Yaskawa INFORM job: CONTOUR.JBI

/JOB
//NAME CONTOUR
//POS
///NPOS 1076,0,0,0,0,0
///TOOL 0
///POSTYPE PULSE
///PULSE
C00000=-2822,58859,-1118,-1041,-34109,-89
C00001=-2184,59252,651,-1119,-34320,-350
C00002=-2184,59252,-549,-1119,-34320,-350
C00003=-2209,59236,-572,-1116,-34311,-340
C00004=-2228,59203,-624,-1114,-34290,-332
C00005=-2241,59164,-682,-1113,-34266,-326
C00006=-2250,59123,-744,-1112,-34241,-322
C00007=-2256,59080,-810,-1112,-34215,-319
C00008=-2257,59034,-879,-1113,-34187,-318
C00009=-2256,58989,-948,-1113,-34159,-318
C00010=-2251,58945,-1015,-1115,-34132,-319
C00011=-2245,58902,-1080,-1116,-34106,-321
C00012=-2233,58862,-1139,-1118,-34082,-326
C00013=-2213,58831,-1186,-1122,-34063,-333
C00014=-2187,58817,-1207,-1125,-34055,-343
C00015=-2161,58829,-1188,-1128,-34062,-354
C00016=-2142,58860,-1141,-1130,-34081,-362
C00017=-2133,58899,-1082,-1131,-34105,-367
C00018=-2146,58931,-1034,-1129,-34125,-362
C00019=-2150,58886,-1101,-1129,-34097,-359
C00020=-2165,58851,-1155,-1127,-34076,-353
C00021=-2191,58837,-1177,-1124,-34067,-342
C00022=-2215,58858,-1145,-1121,-34080,-333
C00023=-2231,58895,-1089,-1118,-34102,-327
C00024=-2239,58937,-1026,-1116,-34128,-324
C00025=-2243,58981,-959,-1115,-34155,-323
C00026=-2246,59026,-891,-1114,-34182,-322
C00027=-2245,59072,-822,-1113,-34210,-323
C00028=-2239,59115,-756,-1114,-34237,-326
C00029=-2230,59156,-694,-1114,-34261,-331
C00030=-2215,59193,-638,-1115,-34284,-337
C00031=-2195,59225,-590,-1118,-34304,-346
C00032=-2168,59227,-586,-1121,-34305,-357
C00033=-2143,59211,-610,-1125,-34296,-367
C00034=-2134,59169,-673,-1126,-34270,-369
C00035=-2128,59126,-737,-1128,-34244,-371
C00036=-2125,59081,-805,-1129,-34217,-372
C00037=-2109,59103,-772,-1131,-34230,-379
C00038=-2115,59146,-707,-1129,-34256,-377
C00039=-2123,59188,-644,-1128,-34282,-374
C00040=-2131,59230,-580,-1126,-34307,-372
C00041=-2155,59248,-554,-1122,-34318,-362
C00042=-2184,59252,-549,-1119,-34320,-350
C00043=-2184,59252,651,-1119,-34320,-350
C00044=-1874,59033,327,-1163,-34189,-472
C00045=-1874,59033,-873,-1163,-34189,-472
C00046=-1891,59025,-886,-1161,-34184,-465
C00047=-1906,59007,-912,-1159,-34173,-459
C00048=-1916,58983,-950,-1158,-34158,-455
C00049=-1926,58964,-979,-1157,-34146,-450
C00050=-1930,58992,-936,-1156,-34164,-449
C00051=-1936,59020,-895,-1155,-34180,-447
C00052=-1949,59030,-879,-1153,-34186,-442
C00053=-1949,59002,-922,-1153,-34169,-442
C00054=-1942,58975,-962,-1155,-34153,-444
C00055=-1936,58948,-1003,-1156,-34136,-446
C00056=-1933,58919,-1047,-1157,-34119,-447
C00057=-1930,58890,-1091,-1158,-34101,-448
C00058=-1928,58860,-1136,-1158,-34083,-448
C00059=-1925,58831,-1180,-1159,-34065,-449
C00060=-1914,58811,-1211,-1161,-34052,-453
C00061=-1907,58835,-1174,-1162,-34067,-456
C00062=-1911,58864,-1130,-1161,-34085,-455
C00063=-1912,58893,-1086,-1160,-34103,-455
C00064=-1913,58924,-1039,-1159,-34122,-455
C00065=-1911,58952,-997,-1159,-34139,-457
C00066=-1904,58978,-957,-1160,-34155,-460
C00067=-1892,59001,-922,-1161,-34169,-465
C00068=-1875,59009,-909,-1163,-34175,-472
C00069=-1858,59003,-918,-1165,-34171,-479
C00070=-1844,58981,-950,-1167,-34158,-484
C00071=-1834,58957,-988,-1169,-34142,-487
C00072=-1828,58930,-1029,-1170,-34126,-490
C00073=-1822,58902,-1070,-1172,-34109,-492
C00074=-1819,58873,-1114,-1173,-34092,-493
C00075=-1818,58843,-1160,-1173,-34073,-493
C00076=-1806,58826,-1186,-1175,-34063,-497
C00077=-1798,58850,-1149,-1176,-34078,-500
C00078=-1803,58878,-1107,-1175,-34095,-499
C00079=-1810,58905,-1066,-1173,-34111,-497
C00080=-1814,58933,-1023,-1172,-34128,-495
C00081=-1821,58960,-983,-1171,-34145,-493
C00082=-1830,58986,-944,-1169,-34160,-490
C00083=-1841,59009,-908,-1167,-34175,-485
C00084=-1856,59028,-880,-1165,-34186,-480
C00085=-1874,59033,-873,-1163,-34189,-472
C00086=-1874,59033,327,-1163,-34189,-472
C00087=-1240,59056,376,-1245,-34208,-728
C00088=-1240,59056,-824,-1245,-34208,-728
C00089=-1239,59026,-870,-1246,-34189,-728
C00090=-1230,58999,-911,-1247,-34173,-731
C00091=-1224,58970,-954,-1249,-34155,-733
C00092=-1220,58941,-999,-1250,-34137,-734
C00093=-1215,58911,-1044,-1251,-34119,-736
C00094=-1214,58881,-1090,-1252,-34100,-736
C00095=-1216,58849,-1139,-1252,-34081,-735
C00096=-1220,58819,-1183,-1252,-34062,-733
C00097=-1232,58796,-1220,-1251,-34048,-728
C00098=-1251,58791,-1227,-1248,-34045,-720
C00099=-1268,58804,-1208,-1246,-34053,-713
C00100=-1284,58821,-1182,-1244,-34063,-707
C00101=-1298,58844,-1148,-1241,-34077,-702
C00102=-1307,58870,-1108,-1240,-34093,-698
C00103=-1313,58899,-1064,-1238,-34111,-696
C00104=-1318,58929,-1019,-1237,-34129,-695
C00105=-1321,58959,-973,-1236,-34148,-694
C00106=-1321,58991,-925,-1236,-34167,-694
C00107=-1335,59000,-910,-1234,-34173,-689
C00108=-1336,58972,-953,-1234,-34156,-688
C00109=-1333,58942,-999,-1235,-34137,-689
C00110=-1329,58912,-1045,-1236,-34119,-690
C00111=-1325,58882,-1090,-1237,-34101,-691
C00112=-1319,58854,-1133,-1238,-34083,-693
C00113=-1307,58828,-1172,-1240,-34067,-698
C00114=-1294,58805,-1207,-1242,-34053,-703
C00115=-1278,58788,-1233,-1245,-34043,-709
C00116=-1261,58774,-1254,-1247,-34034,-715
C00117=-1243,58771,-1258,-1250,-34032,-723
C00118=-1224,58777,-1248,-1252,-34036,-730
C00119=-1211,58799,-1214,-1253,-34050,-736
C00120=-1204,58827,-1171,-1254,-34067,-739
C00121=-1202,58859,-1123,-1254,-34087,-740
C00122=-1201,58890,-1075,-1253,-34106,-741
C00123=-1204,58920,-1029,-1252,-34125,-740
C00124=-1208,58951,-983,-1251,-34143,-739
C00125=-1213,58980,-939,-1250,-34161,-738
C00126=-1219,59008,-896,-1249,-34179,-736
C00127=-1227,59036,-854,-1247,-34196,-733
C00128=-1240,59056,-824,-1245,-34208,-728
C00129=-1240,59056,376,-1245,-34208,-728
C00130=-2046,59034,324,-1140,-34188,-403
C00131=-2046,59034,-876,-1140,-34188,-403
C00132=-2039,59033,-876,-1141,-34188,-406
C00133=-2033,59026,-888,-1142,-34183,-408
C00134=-2027,59017,-900,-1143,-34178,-411
C00135=-2021,59011,-910,-1144,-34174,-413
C00136=-2016,59002,-923,-1145,-34169,-415
C00137=-2013,58991,-940,-1145,-34162,-416
C00138=-2012,58979,-958,-1145,-34155,-416
C00139=-2012,58967,-976,-1146,-34148,-416
C00140=-2014,58955,-994,-1146,-34141,-415
C00141=-2013,58943,-1012,-1146,-34133,-415
C00142=-2014,58931,-1030,-1146,-34126,-415
C00143=-2015,58918,-1050,-1146,-34118,-414
C00144=-2016,58906,-1068,-1146,-34110,-414
C00145=-2017,58894,-1086,-1146,-34103,-413
C00146=-2020,58883,-1104,-1146,-34096,-412
C00147=-2024,58873,-1119,-1146,-34090,-410
C00148=-2029,58864,-1133,-1145,-34084,-408
C00149=-2035,58856,-1144,-1145,-34080,-405
C00150=-2042,58853,-1149,-1144,-34078,-402
C00151=-2050,58852,-1151,-1143,-34077,-399
C00152=-2057,58856,-1144,-1142,-34080,-396
C00153=-2064,58859,-1140,-1141,-34081,-394
C00154=-2070,58867,-1128,-1140,-34086,-391
C00155=-2076,58874,-1118,-1139,-34090,-389
C00156=-2081,58884,-1103,-1138,-34097,-387
C00157=-2084,58895,-1086,-1137,-34103,-386
C00158=-2087,58906,-1069,-1137,-34110,-385
C00159=-2087,58919,-1051,-1137,-34118,-385
C00160=-2088,58931,-1032,-1136,-34125,-385
C00161=-2087,58943,-1014,-1136,-34132,-385
C00162=-2086,58955,-996,-1136,-34140,-386
C00163=-2083,58966,-979,-1136,-34146,-387
C00164=-2080,58977,-963,-1137,-34153,-389
C00165=-2078,58988,-946,-1137,-34160,-390
C00166=-2074,58998,-930,-1137,-34166,-392
C00167=-2070,59007,-916,-1137,-34172,-393
C00168=-2066,59017,-901,-1138,-34178,-395
C00169=-2060,59025,-890,-1139,-34183,-398
C00170=-2053,59029,-883,-1139,-34185,-400
C00171=-2046,59034,-876,-1140,-34188,-403
C00172=-2046,59034,324,-1140,-34188,-403
C00173=-1405,59028,330,-1224,-34190,-661
C00174=-1405,59028,-870,-1224,-34190,-661
C00175=-1398,59001,-912,-1226,-34173,-664
C00176=-1386,58977,-947,-1228,-34159,-668
C00177=-1375,58952,-985,-1229,-34143,-672
C00178=-1368,58924,-1027,-1231,-34126,-674
C00179=-1363,58896,-1070,-1232,-34109,-676
C00180=-1359,58866,-1115,-1233,-34090,-677
C00181=-1361,58835,-1163,-1233,-34071,-676
C00182=-1371,58810,-1201,-1232,-34056,-672
C00183=-1389,58802,-1213,-1230,-34051,-664
C00184=-1407,58808,-1204,-1228,-34054,-657
C00185=-1423,58827,-1176,-1225,-34066,-651
C00186=-1433,58852,-1138,-1223,-34081,-647
C00187=-1442,58879,-1098,-1222,-34098,-644
C00188=-1445,58909,-1052,-1221,-34116,-643
C00189=-1443,58939,-1006,-1221,-34135,-645
C00190=-1434,58965,-966,-1221,-34151,-649
C00191=-1419,58984,-938,-1223,-34162,-655
C00192=-1405,58980,-943,-1225,-34160,-661
C00193=-1415,59003,-908,-1223,-34174,-657
C00194=-1433,58997,-917,-1221,-34170,-649
C00195=-1448,58976,-949,-1219,-34158,-643
C00196=-1456,58950,-990,-1219,-34141,-640
C00197=-1460,58920,-1035,-1219,-34123,-638
C00198=-1459,58889,-1082,-1220,-34104,-638
C00199=-1453,58861,-1125,-1221,-34086,-640
C00200=-1442,58835,-1164,-1223,-34071,-643
C00201=-1432,58810,-1203,-1224,-34055,-647
C00202=-1417,58791,-1231,-1227,-34044,-653
C00203=-1399,58782,-1244,-1229,-34038,-660
C00204=-1380,58781,-1245,-1232,-34038,-668
C00205=-1362,58792,-1229,-1234,-34044,-675
C00206=-1352,58816,-1192,-1235,-34059,-680
C00207=-1347,58845,-1147,-1235,-34077,-682
C00208=-1348,58876,-1100,-1234,-34097,-682
C00209=-1352,58906,-1055,-1233,-34115,-681
C00210=-1358,58934,-1013,-1232,-34132,-679
C00211=-1365,58961,-971,-1230,-34149,-676
C00212=-1376,58986,-933,-1229,-34164,-672
C00213=-1389,59010,-897,-1226,-34179,-667
C00214=-1405,59028,-870,-1224,-34190,-661
C00215=-1405,59028,330,-1224,-34190,-661
C00216=-2050,59056,358,-1139,-34202,-402
C00217=-2050,59056,-842,-1139,-34202,-402
C00218=-2062,59047,-855,-1138,-34196,-397
C00219=-2072,59034,-875,-1137,-34188,-393
C00220=-2082,59018,-900,-1136,-34179,-389
C00221=-2088,59000,-927,-1135,-34168,-386
C00222=-2094,58982,-956,-1135,-34156,-383
C00223=-2098,58962,-986,-1135,-34144,-381
C00224=-2101,58941,-1017,-1135,-34131,-380
C00225=-2100,58919,-1050,-1135,-34118,-380
C00226=-2097,58899,-1081,-1136,-34105,-381
C00227=-2093,58879,-1111,-1137,-34093,-382
C00228=-2086,58861,-1139,-1138,-34082,-385
C00229=-2075,58850,-1155,-1139,-34075,-389
C00230=-2064,58840,-1170,-1141,-34070,-394
C00231=-2051,58834,-1178,-1143,-34066,-399
C00232=-2037,58836,-1176,-1145,-34067,-404
C00233=-2025,58842,-1165,-1146,-34071,-409
C00234=-2014,58856,-1144,-1147,-34080,-414
C00235=-2008,58874,-1116,-1148,-34091,-416
C00236=-2004,58894,-1086,-1148,-34103,-418
C00237=-2002,58916,-1053,-1148,-34116,-419
C00238=-1995,58905,-1069,-1149,-34110,-422
C00239=-1990,58886,-1098,-1150,-34098,-424
C00240=-1986,58866,-1128,-1151,-34086,-425
C00241=-1983,58846,-1159,-1152,-34074,-426
C00242=-1976,58829,-1185,-1153,-34063,-429
C00243=-1963,58829,-1185,-1154,-34063,-434
C00244=-1965,58848,-1156,-1154,-34075,-433
C00245=-1972,58866,-1128,-1153,-34086,-431
C00246=-1976,58886,-1098,-1152,-34098,-430
C00247=-1980,58906,-1068,-1151,-34110,-428
C00248=-1984,58926,-1038,-1150,-34123,-427
C00249=-1989,58945,-1009,-1149,-34134,-425
C00250=-1992,58966,-978,-1148,-34147,-424
C00251=-1995,58986,-947,-1148,-34159,-423
C00252=-1999,59006,-917,-1147,-34171,-422
C00253=-2004,59025,-888,-1146,-34183,-420
C00254=-2016,59026,-887,-1144,-34184,-415
C00255=-2026,59042,-863,-1143,-34193,-411
C00256=-2036,59055,-843,-1141,-34201,-407
C00257=-2050,59056,-842,-1139,-34202,-402
C00258=-2050,59056,358,-1139,-34202,-402
C00259=-1609,59068,387,-1197,-34213,-579
C00260=-1609,59068,-813,-1197,-34213,-579
C00261=-1614,59016,-893,-1197,-34180,-577
C00262=-1610,58960,-979,-1199,-34146,-578
C00263=-1598,58908,-1057,-1201,-34114,-582
C00264=-1580,58861,-1128,-1204,-34086,-588
C00265=-1547,58852,-1140,-1209,-34080,-602
C00266=-1529,58898,-1070,-1210,-34109,-609
C00267=-1527,58953,-987,-1209,-34143,-611
C00268=-1514,58951,-990,-1211,-34141,-616
C00269=-1493,58905,-1060,-1215,-34113,-624
C00270=-1475,58856,-1132,-1218,-34084,-631
C00271=-1464,58804,-1212,-1220,-34051,-634
C00272=-1466,58747,-1298,-1221,-34016,-633
C00273=-1481,58698,-1373,-1220,-33986,-626
C00274=-1503,58656,-1438,-1218,-33960,-617
C00275=-1534,58636,-1468,-1214,-33948,-604
C00276=-1565,58661,-1431,-1210,-33963,-592
C00277=-1589,58705,-1365,-1206,-33990,-582
C00278=-1608,58752,-1293,-1202,-34019,-576
C00279=-1616,58761,-1281,-1201,-34024,-573
C00280=-1600,58711,-1356,-1204,-33993,-578
C00281=-1579,58665,-1425,-1208,-33965,-586
C00282=-1553,58628,-1481,-1212,-33943,-596
C00283=-1518,58620,-1493,-1216,-33938,-610
C00284=-1488,58646,-1453,-1220,-33954,-623
C00285=-1467,58690,-1385,-1222,-33981,-632
C00286=-1453,58740,-1309,-1223,-34012,-638
C00287=-1451,58795,-1225,-1222,-34046,-640
C00288=-1458,58849,-1143,-1220,-34079,-637
C00289=-1474,58899,-1068,-1217,-34109,-632
C00290=-1493,58945,-998,-1214,-34138,-625
C00291=-1515,58990,-930,-1210,-34166,-616
C00292=-1534,59037,-860,-1207,-34194,-610
C00293=-1544,59007,-905,-1206,-34176,-605
C00294=-1538,58952,-989,-1208,-34142,-606
C00295=-1540,58896,-1073,-1209,-34108,-605
C00296=-1564,58871,-1113,-1206,-34092,-595
C00297=-1585,58912,-1050,-1203,-34117,-587
C00298=-1595,58965,-970,-1200,-34150,-584
C00299=-1599,59022,-884,-1199,-34184,-583
C00300=-1609,59068,-813,-1197,-34213,-579
C00301=-1609,59068,387,-1197,-34213,-579
C00302=-3014,58953,182,-1015,-34132,-13
C00303=-3014,58953,-1018,-1015,-34132,-13
C00304=-3024,58937,-1043,-1014,-34122,-9
C00305=-3030,58917,-1073,-1013,-34110,-6
C00306=-3034,58895,-1106,-1013,-34097,-4
C00307=-3037,58873,-1140,-1013,-34083,-3
C00308=-3040,58850,-1174,-1013,-34070,-1
C00309=-3044,58828,-1207,-1013,-34057,1
C00310=-3046,58805,-1242,-1013,-34043,2
C00311=-3047,58782,-1277,-1013,-34028,3
C00312=-3049,58758,-1312,-1013,-34014,4
C00313=-3050,58734,-1349,-1013,-34000,4
C00314=-3050,58712,-1383,-1013,-33986,5
C00315=-3048,58689,-1417,-1014,-33972,4
C00316=-3047,58666,-1452,-1015,-33958,4
C00317=-3043,58644,-1484,-1015,-33945,3
C00318=-3037,58624,-1515,-1016,-33933,1
C00319=-3031,58604,-1545,-1018,-33921,-2
C00320=-3021,58586,-1571,-1019,-33910,-5
C00321=-3009,58576,-1587,-1021,-33904,-10
C00322=-2996,58566,-1601,-1023,-33898,-15
C00323=-2983,58561,-1609,-1025,-33895,-21
C00324=-2970,58570,-1595,-1026,-33901,-26
C00325=-2959,58584,-1573,-1027,-33909,-30
C00326=-2955,58606,-1541,-1028,-33922,-32
C00327=-2952,58628,-1507,-1028,-33936,-34
C00328=-2946,58649,-1475,-1028,-33948,-36
C00329=-2946,58673,-1439,-1028,-33963,-37
C00330=-2948,58696,-1405,-1027,-33977,-36
C00331=-2950,58719,-1370,-1027,-33991,-36
C00332=-2952,58740,-1339,-1026,-34003,-35
C00333=-2953,58763,-1303,-1025,-34018,-35
C00334=-2957,58785,-1271,-1025,-34031,-34
C00335=-2961,58806,-1239,-1024,-34044,-32
C00336=-2965,58828,-1206,-1023,-34057,-31
C00337=-2969,58849,-1174,-1022,-34070,-29
C00338=-2972,58871,-1141,-1021,-34083,-28
C00339=-2983,58885,-1120,-1020,-34091,-24
C00340=-2991,58903,-1093,-1018,-34102,-21
C00341=-2996,58924,-1061,-1017,-34115,-20
C00342=-3001,58944,-1032,-1016,-34127,-18
C00343=-3014,58953,-1018,-1015,-34132,-13
C00344=-3014,58953,182,-1015,-34132,-13
C00345=-2663,58940,170,-1061,-34127,-154
C00346=-2663,58940,-1030,-1061,-34127,-154
C00347=-2675,58925,-1053,-1060,-34118,-149
C00348=-2682,58905,-1084,-1059,-34105,-145
C00349=-2691,58886,-1113,-1058,-34094,-142
C00350=-2696,58863,-1147,-1058,-34080,-140
C00351=-2699,58840,-1183,-1058,-34065,-138
C00352=-2702,58816,-1219,-1058,-34051,-137
C00353=-2705,58792,-1254,-1058,-34037,-135
C00354=-2707,58769,-1290,-1058,-34022,-134
C00355=-2709,58744,-1327,-1058,-34007,-133
C00356=-2710,58719,-1365,-1058,-33992,-132
C00357=-2710,58693,-1404,-1058,-33977,-132
C00358=-2707,58671,-1438,-1059,-33963,-133
C00359=-2700,58649,-1470,-1060,-33950,-135
C00360=-2696,58627,-1504,-1061,-33936,-137
C00361=-2690,58605,-1537,-1062,-33923,-139
C00362=-2684,58584,-1569,-1064,-33910,-141
C00363=-2677,58563,-1601,-1065,-33897,-143
C00364=-2668,58543,-1630,-1066,-33885,-147
C00365=-2658,58524,-1659,-1068,-33874,-150
C00366=-2645,58514,-1674,-1070,-33868,-156
C00367=-2631,58520,-1665,-1072,-33871,-161
C00368=-2623,58540,-1635,-1072,-33883,-165
C00369=-2617,58561,-1603,-1073,-33896,-168
C00370=-2611,58582,-1570,-1073,-33910,-170
C00371=-2608,58606,-1534,-1073,-33924,-172
C00372=-2608,58631,-1496,-1073,-33939,-172
C00373=-2607,58657,-1457,-1073,-33955,-173
C00374=-2608,58681,-1420,-1072,-33970,-173
C00375=-2609,58706,-1383,-1072,-33985,-173
C00376=-2611,58730,-1347,-1071,-33999,-172
C00377=-2614,58753,-1312,-1070,-34013,-171
C00378=-2617,58776,-1277,-1069,-34027,-170
C00379=-2620,58799,-1242,-1069,-34041,-169
C00380=-2625,58822,-1208,-1068,-34055,-168
C00381=-2628,58845,-1174,-1067,-34069,-167
C00382=-2632,58868,-1139,-1066,-34083,-165
C00383=-2638,58889,-1107,-1065,-34096,-163
C00384=-2644,58911,-1075,-1064,-34109,-161
C00385=-2650,58932,-1042,-1063,-34122,-159
C00386=-2663,58940,-1030,-1061,-34127,-154
C00387=-2663,58940,170,-1061,-34127,-154
C00388=-2757,59223,596,-1044,-34298,-119
C00389=-2757,59223,-604,-1044,-34298,-119
C00390=-2693,59208,-626,-1053,-34290,-145
C00391=-2630,59182,-664,-1061,-34274,-170
C00392=-2574,59133,-737,-1069,-34245,-192
C00393=-2526,59062,-843,-1077,-34202,-210
C00394=-2480,58986,-957,-1084,-34156,-228
C00395=-2446,58899,-1088,-1090,-34103,-240
C00396=-2419,58806,-1228,-1095,-34047,-250
C00397=-2407,58704,-1382,-1098,-33985,-254
C00398=-2398,58601,-1538,-1101,-33922,-256
C00399=-2407,58496,-1697,-1101,-33858,-251
C00400=-2428,58399,-1844,-1100,-33799,-241
C00401=-2458,58309,-1981,-1098,-33744,-228
C00402=-2493,58223,-2111,-1094,-33691,-213
C00403=-2541,58152,-2220,-1089,-33648,-193
C00404=-2597,58101,-2298,-1083,-33616,-170
C00405=-2656,58061,-2359,-1075,-33592,-146
C00406=-2720,58047,-2380,-1067,-33584,-120
C00407=-2787,58043,-2387,-1058,-33581,-93
C00408=-2853,58050,-2378,-1049,-33585,-66
C00409=-2917,58074,-2342,-1041,-33600,-41
C00410=-2978,58104,-2299,-1032,-33618,-17
C00411=-3037,58144,-2238,-1024,-33642,6
C00412=-3091,58201,-2154,-1016,-33677,27
C00413=-3135,58277,-2039,-1009,-33723,44
C00414=-3171,58365,-1907,-1003,-33776,57
C00415=-3195,58460,-1765,-998,-33833,66
C00416=-3207,58561,-1612,-995,-33894,70
C00417=-3212,58668,-1452,-993,-33959,70
C00418=-3203,58772,-1294,-992,-34022,66
C00419=-3186,58872,-1144,-993,-34082,58
C00420=-3163,58967,-999,-995,-34140,47
C00421=-3125,59052,-871,-999,-34191,31
C00422=-3079,59128,-755,-1003,-34238,12
C00423=-3024,59183,-671,-1010,-34272,-11
C00424=-2964,59218,-617,-1017,-34293,-36
C00425=-2901,59212,-624,-1026,-34290,-61
C00426=-2922,59190,-659,-1023,-34277,-53
C00427=-2857,59192,-654,-1032,-34278,-79
C00428=-2823,59217,-616,-1036,-34294,-92
C00429=-2757,59223,-604,-1044,-34298,-119
C00430=-2757,59223,596,-1044,-34298,-119
C00431=-1081,58531,-419,-1275,-33885,-784
C00432=-1081,58531,-1619,-1275,-33885,-784
C00433=-1082,58530,-1621,-1275,-33885,-784
C00434=-1083,58529,-1623,-1275,-33884,-784
C00435=-1084,58528,-1624,-1275,-33883,-783
C00436=-1084,58527,-1626,-1275,-33883,-783
C00437=-1085,58525,-1628,-1275,-33882,-783
C00438=-1085,58524,-1631,-1275,-33881,-783
C00439=-1085,58522,-1633,-1275,-33880,-783
C00440=-1085,58520,-1636,-1275,-33879,-783
C00441=-1085,58519,-1638,-1275,-33878,-783
C00442=-1084,58518,-1640,-1275,-33877,-783
C00443=-1083,58518,-1640,-1275,-33877,-784
C00444=-1082,58516,-1642,-1275,-33876,-784
C00445=-1081,58515,-1644,-1276,-33875,-784
C00446=-1080,58514,-1646,-1276,-33875,-784
C00447=-1080,58513,-1647,-1276,-33874,-785
C00448=-1079,58512,-1649,-1276,-33873,-785
C00449=-1078,58511,-1649,-1276,-33873,-785
C00450=-1077,58511,-1649,-1276,-33873,-786
C00451=-1076,58511,-1649,-1276,-33873,-786
C00452=-1075,58511,-1649,-1277,-33873,-787
C00453=-1074,58512,-1649,-1277,-33873,-787
C00454=-1073,58513,-1647,-1277,-33874,-787
C00455=-1073,58515,-1644,-1277,-33875,-788
C00456=-1073,58516,-1642,-1277,-33876,-788
C00457=-1072,58518,-1640,-1277,-33877,-788
C00458=-1071,58519,-1638,-1277,-33878,-788
C00459=-1071,58521,-1635,-1277,-33879,-788
C00460=-1071,58522,-1632,-1277,-33880,-788
C00461=-1071,58524,-1630,-1277,-33881,-788
C00462=-1072,58526,-1628,-1277,-33882,-788
C00463=-1073,58527,-1626,-1277,-33883,-788
C00464=-1073,58528,-1624,-1276,-33883,-787
C00465=-1074,58529,-1622,-1276,-33884,-787
C00466=-1075,58531,-1620,-1276,-33885,-787
C00467=-1076,58531,-1619,-1276,-33885,-787
C00468=-1077,58531,-1619,-1276,-33885,-786
C00469=-1078,58531,-1619,-1276,-33885,-786
C00470=-1079,58531,-1619,-1276,-33885,-785
C00471=-1080,58531,-1619,-1275,-33885,-785
C00472=-1081,58531,-1619,-1275,-33885,-784
C00473=-1081,58531,-419,-1275,-33885,-784
C00474=-742,58586,-329,-1319,-33921,-922
C00475=-742,58586,-1529,-1319,-33921,-922
C00476=-756,58577,-1543,-1317,-33916,-916
C00477=-771,58570,-1554,-1315,-33911,-909
C00478=-786,58561,-1567,-1314,-33906,-903
C00479=-799,58547,-1590,-1312,-33896,-898
C00480=-807,58525,-1624,-1312,-33883,-895
C00481=-795,58511,-1645,-1313,-33874,-899
C00482=-788,58532,-1612,-1314,-33888,-902
C00483=-774,58545,-1592,-1315,-33896,-908
C00484=-760,58555,-1576,-1317,-33902,-914
C00485=-744,58563,-1565,-1319,-33907,-920
C00486=-728,58563,-1564,-1321,-33907,-927
C00487=-714,58552,-1581,-1323,-33900,-932
C00488=-708,58528,-1617,-1324,-33885,-935
C00489=-708,58503,-1656,-1325,-33870,-934
C00490=-711,58477,-1695,-1325,-33854,-932
C00491=-716,58453,-1731,-1325,-33839,-930
C00492=-724,58432,-1764,-1324,-33825,-927
C00493=-731,58410,-1798,-1323,-33812,-923
C00494=-740,58388,-1830,-1323,-33799,-919
C00495=-748,58367,-1864,-1322,-33785,-916
C00496=-756,58345,-1897,-1321,-33772,-912
C00497=-763,58322,-1932,-1321,-33758,-909
C00498=-770,58300,-1966,-1320,-33744,-906
C00499=-771,58277,-2001,-1321,-33730,-905
C00500=-759,58283,-1992,-1322,-33733,-910
C00501=-751,58303,-1961,-1323,-33746,-914
C00502=-746,58327,-1924,-1323,-33761,-916
C00503=-738,58349,-1891,-1324,-33774,-919
C00504=-731,58371,-1857,-1324,-33788,-923
C00505=-721,58392,-1825,-1325,-33801,-927
C00506=-713,58413,-1792,-1326,-33814,-931
C00507=-705,58435,-1759,-1326,-33828,-934
C00508=-700,58458,-1723,-1327,-33842,-937
C00509=-695,58483,-1686,-1327,-33857,-939
C00510=-693,58508,-1647,-1327,-33873,-940
C00511=-694,58535,-1606,-1326,-33890,-940
C00512=-698,58559,-1569,-1325,-33905,-939
C00513=-709,58576,-1543,-1323,-33915,-935
C00514=-724,58585,-1530,-1321,-33921,-929
C00515=-742,58586,-1529,-1319,-33921,-922
C00516=-742,58586,-329,-1319,-33921,-922
C00517=-2202,58626,-297,-1126,-33938,-335
C00518=-2202,58626,-1497,-1126,-33938,-335
C00519=-2202,58576,-1571,-1127,-33908,-335
C00520=-2191,58526,-1647,-1129,-33877,-338
C00521=-2185,58474,-1727,-1131,-33845,-340
C00522=-2209,58452,-1760,-1128,-33832,-330
C00523=-2242,58446,-1769,-1124,-33828,-317
C00524=-2261,58420,-1810,-1122,-33812,-309
C00525=-2228,58429,-1795,-1126,-33818,-322
C00526=-2194,58434,-1787,-1130,-33821,-336
C00527=-2180,58402,-1836,-1133,-33801,-341
C00528=-2179,58346,-1920,-1134,-33767,-341
C00529=-2180,58291,-2003,-1135,-33733,-340
C00530=-2162,58287,-2009,-1137,-33731,-347
C00531=-2165,58342,-1926,-1136,-33764,-346
C00532=-2165,58398,-1842,-1135,-33799,-347
C00533=-2161,58445,-1769,-1135,-33828,-349
C00534=-2129,58457,-1751,-1139,-33835,-362
C00535=-2096,58469,-1732,-1143,-33842,-376
C00536=-2079,58446,-1768,-1145,-33828,-382
C00537=-2073,58393,-1846,-1147,-33796,-384
C00538=-2069,58340,-1928,-1149,-33764,-385
C00539=-2068,58285,-2010,-1149,-33730,-384
C00540=-2053,58268,-2037,-1152,-33719,-390
C00541=-2050,58322,-1954,-1151,-33753,-392
C00542=-2047,58377,-1871,-1151,-33786,-394
C00543=-2040,58428,-1793,-1151,-33818,-398
C00544=-2028,58477,-1719,-1152,-33848,-403
C00545=-2005,58514,-1663,-1154,-33870,-413
C00546=-1981,58518,-1656,-1157,-33873,-422
C00547=-2012,58530,-1638,-1153,-33880,-410
C00548=-2035,58493,-1696,-1151,-33857,-401
C00549=-2048,58445,-1768,-1150,-33828,-395
C00550=-2061,58430,-1791,-1148,-33819,-389
C00551=-2066,58482,-1712,-1147,-33851,-388
C00552=-2084,58498,-1688,-1144,-33860,-381
C00553=-2113,58482,-1712,-1140,-33851,-369
C00554=-2145,58472,-1728,-1136,-33844,-356
C00555=-2171,58479,-1718,-1133,-33848,-346
C00556=-2178,58531,-1639,-1131,-33880,-344
C00557=-2187,58582,-1563,-1129,-33911,-341
C00558=-2202,58626,-1497,-1126,-33938,-335
C00559=-2202,58626,-297,-1126,-33938,-335
C00560=-1361,58593,-331,-1237,-33922,-673
C00561=-1361,58593,-1531,-1237,-33922,-673
C00562=-1359,58521,-1641,-1239,-33877,-673
C00563=-1349,58450,-1747,-1242,-33834,-676
C00564=-1369,58412,-1806,-1240,-33811,-667
C00565=-1394,58398,-1827,-1236,-33802,-657
C00566=-1347,58389,-1840,-1243,-33797,-675
C00567=-1336,58322,-1942,-1246,-33755,-679
C00568=-1332,58248,-2055,-1247,-33710,-679
C00569=-1318,58210,-2112,-1250,-33686,-685
C00570=-1319,58284,-1999,-1248,-33732,-685
C00571=-1326,58356,-1890,-1246,-33776,-683
C00572=-1306,58397,-1828,-1248,-33801,-692
C00573=-1263,58420,-1791,-1253,-33816,-710
C00574=-1243,58376,-1858,-1257,-33789,-717
C00575=-1231,58307,-1963,-1260,-33746,-721
C00576=-1224,58234,-2074,-1262,-33701,-723
C00577=-1208,58190,-2141,-1265,-33674,-729
C00578=-1209,58264,-2029,-1263,-33720,-729
C00579=-1207,58339,-1915,-1262,-33766,-731
C00580=-1185,58401,-1819,-1264,-33805,-741
C00581=-1145,58390,-1836,-1269,-33798,-757
C00582=-1123,58328,-1930,-1273,-33759,-765
C00583=-1111,58258,-2036,-1276,-33716,-768
C00584=-1107,58184,-2149,-1278,-33671,-769
C00585=-1090,58197,-2129,-1280,-33679,-776
C00586=-1099,58268,-2020,-1278,-33723,-774
C00587=-1111,58337,-1915,-1275,-33765,-769
C00588=-1133,58400,-1821,-1271,-33804,-762
C00589=-1173,58432,-1772,-1265,-33824,-746
C00590=-1205,58383,-1848,-1262,-33793,-732
C00591=-1225,58353,-1893,-1260,-33775,-724
C00592=-1236,58423,-1787,-1257,-33818,-720
C00593=-1251,58491,-1684,-1254,-33860,-716
C00594=-1265,58559,-1581,-1251,-33901,-711
C00595=-1277,58545,-1601,-1249,-33893,-706
C00596=-1262,58478,-1704,-1252,-33851,-711
C00597=-1271,58428,-1780,-1252,-33821,-707
C00598=-1316,58415,-1800,-1246,-33813,-688
C00599=-1337,58466,-1723,-1243,-33844,-681
C00600=-1345,58538,-1613,-1241,-33888,-679
C00601=-1361,58593,-1531,-1237,-33922,-673
C00602=-1361,58593,-331,-1237,-33922,-673
C00603=-1734,58518,-452,-1190,-33874,-522
C00604=-1734,58518,-1652,-1190,-33874,-522
C00605=-1749,58511,-1663,-1188,-33870,-515
C00606=-1765,58502,-1676,-1186,-33864,-509
C00607=-1778,58485,-1703,-1184,-33853,-504
C00608=-1785,58461,-1738,-1184,-33839,-500
C00609=-1792,58437,-1775,-1183,-33824,-497
C00610=-1795,58411,-1815,-1183,-33808,-496
C00611=-1798,58384,-1856,-1184,-33792,-494
C00612=-1797,58356,-1898,-1184,-33775,-494
C00613=-1795,58330,-1939,-1185,-33758,-495
C00614=-1788,58306,-1975,-1186,-33744,-497
C00615=-1777,58284,-2008,-1188,-33730,-501
C00616=-1762,58273,-2024,-1190,-33723,-507
C00617=-1745,58268,-2031,-1192,-33721,-514
C00618=-1728,58269,-2029,-1195,-33721,-521
C00619=-1712,58274,-2021,-1197,-33724,-527
C00620=-1697,58286,-2002,-1198,-33732,-534
C00621=-1683,58300,-1981,-1200,-33740,-539
C00622=-1670,58316,-1957,-1202,-33750,-545
C00623=-1684,58311,-1964,-1200,-33747,-539
C00624=-1699,58301,-1981,-1198,-33741,-533
C00625=-1714,58291,-1996,-1196,-33735,-527
C00626=-1731,58287,-2002,-1194,-33732,-520
C00627=-1749,58288,-2001,-1192,-33733,-513
C00628=-1765,58297,-1988,-1189,-33738,-507
C00629=-1775,58316,-1959,-1188,-33750,-502
C00630=-1782,58340,-1922,-1186,-33765,-500
C00631=-1784,58367,-1882,-1186,-33781,-500
C00632=-1783,58395,-1840,-1185,-33798,-501
C00633=-1780,58421,-1799,-1185,-33814,-502
C00634=-1774,58446,-1762,-1186,-33830,-505
C00635=-1766,58469,-1727,-1186,-33844,-508
C00636=-1753,58485,-1701,-1188,-33854,-514
C00637=-1737,58494,-1689,-1190,-33859,-520
C00638=-1720,58493,-1688,-1192,-33859,-527
C00639=-1707,58479,-1710,-1194,-33850,-532
C00640=-1695,58460,-1738,-1196,-33839,-537
C00641=-1693,58476,-1715,-1196,-33848,-538
C00642=-1703,58498,-1681,-1194,-33862,-534
C00643=-1717,58514,-1658,-1192,-33871,-529
C00644=-1734,58518,-1652,-1190,-33874,-522
C00645=-1734,58518,-452,-1190,-33874,-522
C00646=-1907,58498,-485,-1167,-33861,-452
C00647=-1907,58498,-1685,-1167,-33861,-452
C00648=-1898,58500,-1682,-1168,-33862,-456
C00649=-1889,58495,-1689,-1170,-33859,-459
C00650=-1883,58486,-1703,-1171,-33854,-462
C00651=-1882,58471,-1725,-1171,-33845,-462
C00652=-1881,58456,-1748,-1171,-33836,-462
C00653=-1878,58442,-1769,-1172,-33827,-463
C00654=-1877,58428,-1791,-1172,-33818,-463
C00655=-1877,58413,-1813,-1173,-33809,-463
C00656=-1877,58397,-1837,-1173,-33800,-463
C00657=-1876,58383,-1859,-1173,-33791,-463
C00658=-1877,58368,-1881,-1173,-33782,-462
C00659=-1878,58353,-1904,-1173,-33772,-462
C00660=-1879,58338,-1927,-1174,-33763,-461
C00661=-1882,58325,-1947,-1173,-33755,-460
C00662=-1886,58312,-1967,-1173,-33747,-458
C00663=-1892,58301,-1984,-1172,-33740,-455
C00664=-1898,58291,-1999,-1172,-33734,-453
C00665=-1905,58280,-2015,-1171,-33728,-450
C00666=-1914,58274,-2025,-1170,-33724,-446
C00667=-1923,58272,-2028,-1169,-33723,-443
C00668=-1931,58273,-2027,-1168,-33723,-439
C00669=-1939,58280,-2016,-1167,-33728,-436
C00670=-1946,58290,-2001,-1166,-33734,-434
C00671=-1951,58303,-1982,-1165,-33741,-432
C00672=-1956,58315,-1963,-1164,-33749,-430
C00673=-1960,58328,-1944,-1163,-33757,-429
C00674=-1962,58342,-1923,-1163,-33765,-428
C00675=-1963,58357,-1900,-1162,-33774,-428
C00676=-1963,58372,-1877,-1162,-33784,-428
C00677=-1961,58387,-1855,-1162,-33793,-429
C00678=-1960,58401,-1833,-1162,-33802,-430
C00679=-1957,58415,-1812,-1162,-33810,-431
C00680=-1953,58428,-1792,-1162,-33818,-433
C00681=-1947,58439,-1775,-1163,-33825,-435
C00682=-1943,58452,-1755,-1163,-33833,-437
C00683=-1937,58463,-1738,-1164,-33840,-439
C00684=-1930,58472,-1724,-1165,-33845,-443
C00685=-1923,58483,-1708,-1165,-33852,-446
C00686=-1915,58492,-1694,-1166,-33857,-449
C00687=-1907,58498,-1685,-1167,-33861,-452
C00688=-1907,58498,-485,-1167,-33861,-452
C00689=-1595,58512,-458,-1208,-33871,-578
C00690=-1595,58512,-1658,-1208,-33871,-578
C00691=-1619,58496,-1683,-1205,-33861,-568
C00692=-1637,58465,-1731,-1203,-33842,-560
C00693=-1649,58429,-1786,-1202,-33820,-555
C00694=-1658,58390,-1845,-1202,-33796,-551
C00695=-1661,58348,-1908,-1202,-33770,-549
C00696=-1659,58305,-1973,-1203,-33744,-549
C00697=-1651,58266,-2033,-1205,-33720,-552
C00698=-1632,58235,-2079,-1208,-33701,-559
C00699=-1608,58222,-2099,-1211,-33693,-568
C00700=-1582,58214,-2111,-1215,-33688,-579
C00701=-1555,58218,-2104,-1218,-33690,-590
C00702=-1531,58232,-2082,-1221,-33699,-600
C00703=-1511,58262,-2037,-1223,-33718,-608
C00704=-1497,58296,-1984,-1225,-33739,-614
C00705=-1500,58302,-1975,-1224,-33742,-613
C00706=-1519,58272,-2022,-1222,-33724,-605
C00707=-1540,58246,-2061,-1220,-33708,-596
C00708=-1566,58237,-2075,-1217,-33702,-586
C00709=-1593,58237,-2076,-1213,-33702,-575
C00710=-1617,58251,-2055,-1210,-33711,-565
C00711=-1637,58278,-2014,-1206,-33727,-557
C00712=-1648,58316,-1957,-1204,-33750,-554
C00713=-1648,58358,-1893,-1204,-33776,-554
C00714=-1642,58398,-1831,-1204,-33801,-557
C00715=-1632,58437,-1773,-1204,-33825,-562
C00716=-1615,58470,-1723,-1206,-33845,-569
C00717=-1594,58492,-1688,-1209,-33859,-578
C00718=-1568,58487,-1696,-1212,-33856,-588
C00719=-1551,58456,-1743,-1215,-33837,-594
C00720=-1560,58418,-1800,-1214,-33814,-590
C00721=-1585,58409,-1815,-1211,-33808,-580
C00722=-1611,58406,-1819,-1208,-33806,-570
C00723=-1626,58390,-1843,-1206,-33796,-563
C00724=-1599,58388,-1847,-1210,-33795,-574
C00725=-1573,58392,-1839,-1213,-33798,-585
C00726=-1549,58408,-1815,-1216,-33807,-595
C00727=-1538,58444,-1760,-1217,-33830,-600
C00728=-1547,58483,-1701,-1215,-33853,-596
C00729=-1568,58505,-1668,-1212,-33867,-588
C00730=-1595,58512,-1658,-1208,-33871,-578
C00731=-1595,58512,-458,-1208,-33871,-578
C00732=-1905,58524,-446,-1167,-33877,-453
C00733=-1905,58524,-1646,-1167,-33877,-453
C00734=-1920,58516,-1658,-1165,-33872,-447
C00735=-1932,58503,-1678,-1164,-33864,-442
C00736=-1944,58486,-1704,-1163,-33853,-437
C00737=-1954,58468,-1731,-1162,-33843,-433
C00738=-1963,58448,-1762,-1161,-33830,-429
C00739=-1969,58427,-1794,-1160,-33817,-426
C00740=-1974,58404,-1828,-1160,-33803,-424
C00741=-1976,58379,-1866,-1160,-33788,-423
C00742=-1978,58356,-1902,-1160,-33774,-422
C00743=-1975,58332,-1938,-1161,-33759,-423
C00744=-1969,58310,-1972,-1162,-33745,-424
C00745=-1962,58289,-2004,-1164,-33733,-427
C00746=-1951,58270,-2031,-1165,-33721,-431
C00747=-1938,58257,-2051,-1167,-33713,-436
C00748=-1923,58253,-2056,-1169,-33711,-442
C00749=-1909,58256,-2052,-1171,-33713,-448
C00750=-1897,58268,-2033,-1172,-33720,-453
C00751=-1886,58286,-2006,-1174,-33731,-458
C00752=-1875,58304,-1978,-1175,-33742,-462
C00753=-1871,58327,-1944,-1175,-33756,-464
C00754=-1868,58351,-1907,-1175,-33771,-466
C00755=-1862,58368,-1881,-1175,-33782,-468
C00756=-1858,58345,-1917,-1176,-33767,-470
C00757=-1855,58321,-1953,-1177,-33753,-471
C00758=-1850,58298,-1987,-1178,-33739,-472
C00759=-1847,58274,-2023,-1179,-33724,-473
C00760=-1833,58267,-2034,-1181,-33720,-478
C00761=-1825,58281,-2012,-1182,-33729,-482
C00762=-1835,58300,-1984,-1180,-33740,-478
C00763=-1839,58323,-1949,-1179,-33754,-477
C00764=-1843,58346,-1914,-1178,-33768,-476
C00765=-1846,58370,-1878,-1177,-33783,-475
C00766=-1850,58394,-1842,-1177,-33797,-474
C00767=-1853,58417,-1806,-1176,-33812,-473
C00768=-1858,58440,-1772,-1175,-33826,-471
C00769=-1862,58463,-1737,-1174,-33840,-469
C00770=-1869,58485,-1705,-1172,-33853,-467
C00771=-1879,58502,-1679,-1171,-33864,-463
C00772=-1890,58520,-1651,-1169,-33875,-459
C00773=-1905,58524,-1646,-1167,-33877,-453
C00774=-1905,58524,-446,-1167,-33877,-453
C00775=-1082,58453,-539,-1277,-33837,-783
C00776=-1082,58453,-1739,-1277,-33837,-783
C00777=-1087,58442,-1755,-1276,-33830,-781
C00778=-1085,58429,-1776,-1277,-33822,-781
C00779=-1083,58415,-1796,-1277,-33814,-782
C00780=-1079,58402,-1816,-1278,-33805,-783
C00781=-1078,58387,-1838,-1278,-33796,-783
C00782=-1076,58374,-1859,-1279,-33788,-784
C00783=-1074,58360,-1880,-1279,-33779,-785
C00784=-1073,58345,-1902,-1280,-33771,-785
C00785=-1071,58331,-1924,-1280,-33762,-786
C00786=-1067,58319,-1943,-1281,-33754,-787
C00787=-1065,58305,-1964,-1281,-33745,-788
C00788=-1064,58290,-1986,-1282,-33737,-788
C00789=-1063,58276,-2008,-1282,-33728,-788
C00790=-1060,58262,-2029,-1283,-33719,-789
C00791=-1058,58249,-2049,-1283,-33711,-790
C00792=-1056,58235,-2070,-1284,-33702,-790
C00793=-1054,58221,-2091,-1284,-33694,-791
C00794=-1053,58206,-2114,-1285,-33685,-791
C00795=-1051,58192,-2135,-1285,-33676,-792
C00796=-1042,58189,-2139,-1287,-33674,-795
C00797=-1037,58199,-2124,-1287,-33681,-798
C00798=-1036,58213,-2102,-1287,-33689,-798
C00799=-1040,58226,-2083,-1286,-33697,-797
C00800=-1042,58240,-2062,-1286,-33705,-796
C00801=-1044,58254,-2042,-1285,-33714,-795
C00802=-1047,58267,-2021,-1285,-33722,-794
C00803=-1049,58281,-2000,-1284,-33731,-794
C00804=-1050,58295,-1978,-1284,-33740,-794
C00805=-1051,58310,-1956,-1283,-33749,-793
C00806=-1053,58324,-1935,-1283,-33757,-793
C00807=-1056,58337,-1914,-1282,-33766,-792
C00808=-1059,58351,-1894,-1281,-33774,-791
C00809=-1060,58365,-1872,-1281,-33783,-790
C00810=-1062,58379,-1851,-1281,-33791,-790
C00811=-1065,58392,-1830,-1280,-33800,-789
C00812=-1067,58406,-1809,-1279,-33808,-788
C00813=-1069,58420,-1789,-1279,-33817,-788
C00814=-1072,58434,-1768,-1278,-33825,-787
C00815=-1075,58447,-1748,-1278,-33833,-786
C00816=-1082,58453,-1739,-1277,-33837,-783
C00817=-1082,58453,-539,-1277,-33837,-783
C00818=-965,58468,-514,-1292,-33847,-830
C00819=-965,58468,-1714,-1292,-33847,-830
C00820=-991,58457,-1730,-1288,-33840,-820
C00821=-1014,58432,-1768,-1286,-33825,-810
C00822=-1026,58395,-1826,-1285,-33801,-804
C00823=-1020,58352,-1891,-1287,-33775,-806
C00824=-1000,58324,-1933,-1290,-33758,-814
C00825=-972,58315,-1947,-1293,-33752,-825
C00826=-944,58309,-1955,-1297,-33749,-836
C00827=-917,58302,-1966,-1301,-33744,-847
C00828=-891,58286,-1989,-1305,-33735,-857
C00829=-875,58252,-2041,-1308,-33714,-863
C00830=-880,58209,-2106,-1308,-33687,-860
C00831=-899,58177,-2155,-1306,-33667,-852
C00832=-923,58157,-2187,-1303,-33654,-842
C00833=-951,58151,-2196,-1299,-33651,-831
C00834=-974,58174,-2161,-1296,-33665,-822
C00835=-985,58214,-2101,-1294,-33690,-819
C00836=-994,58240,-2062,-1292,-33706,-815
C00837=-992,58196,-2128,-1293,-33679,-815
C00838=-981,58157,-2187,-1295,-33654,-819
C00839=-959,58132,-2225,-1299,-33639,-828
C00840=-930,58129,-2229,-1302,-33637,-839
C00841=-905,58144,-2206,-1305,-33647,-850
C00842=-882,58169,-2168,-1308,-33662,-859
C00843=-867,58205,-2113,-1309,-33684,-866
C00844=-861,58247,-2048,-1309,-33711,-869
C00845=-872,58287,-1987,-1307,-33735,-865
C00846=-894,58313,-1948,-1304,-33751,-856
C00847=-921,58324,-1932,-1300,-33758,-846
C00848=-949,58331,-1921,-1296,-33762,-835
C00849=-977,58335,-1916,-1292,-33764,-823
C00850=-1002,58352,-1890,-1289,-33775,-814
C00851=-1011,58393,-1829,-1287,-33800,-810
C00852=-996,58427,-1776,-1288,-33821,-817
C00853=-970,58442,-1752,-1291,-33831,-828
C00854=-943,58435,-1763,-1295,-33827,-839
C00855=-921,58409,-1803,-1299,-33810,-847
C00856=-904,58394,-1825,-1301,-33801,-854
C00857=-915,58434,-1765,-1299,-33826,-850
C00858=-937,58458,-1728,-1296,-33841,-841
C00859=-965,58468,-1714,-1292,-33847,-830
C00860=-965,58468,-514,-1292,-33847,-830
C00861=-2883,58398,-654,-1040,-33796,-59
C00862=-2883,58398,-1854,-1040,-33796,-59
C00863=-2892,58389,-1867,-1039,-33791,-55
C00864=-2894,58370,-1896,-1039,-33779,-54
C00865=-2891,58352,-1923,-1040,-33768,-55
C00866=-2884,58336,-1947,-1041,-33759,-58
C00867=-2878,58319,-1973,-1042,-33748,-60
C00868=-2872,58303,-1997,-1043,-33739,-62
C00869=-2863,58289,-2017,-1044,-33731,-65
C00870=-2854,58277,-2036,-1046,-33723,-69
C00871=-2844,58267,-2050,-1047,-33717,-73
C00872=-2833,58261,-2060,-1049,-33713,-77
C00873=-2820,58259,-2062,-1051,-33712,-82
C00874=-2807,58259,-2062,-1052,-33712,-87
C00875=-2796,58264,-2054,-1054,-33715,-92
C00876=-2785,58271,-2044,-1055,-33719,-96
C00877=-2775,58279,-2031,-1056,-33724,-101
C00878=-2764,58288,-2017,-1058,-33730,-105
C00879=-2755,58301,-1998,-1059,-33738,-109
C00880=-2746,58315,-1976,-1060,-33747,-113
C00881=-2737,58329,-1955,-1061,-33755,-116
C00882=-2729,58344,-1932,-1061,-33764,-120
C00883=-2722,58360,-1908,-1062,-33774,-123
C00884=-2726,58377,-1882,-1061,-33784,-122
C00885=-2736,58370,-1893,-1060,-33780,-117
C00886=-2745,58356,-1915,-1059,-33771,-114
C00887=-2753,58341,-1937,-1058,-33762,-110
C00888=-2763,58327,-1958,-1057,-33754,-106
C00889=-2771,58313,-1980,-1056,-33745,-103
C00890=-2781,58301,-1998,-1055,-33738,-99
C00891=-2791,58291,-2014,-1054,-33732,-94
C00892=-2802,58286,-2021,-1053,-33729,-90
C00893=-2815,58285,-2023,-1051,-33728,-85
C00894=-2827,58287,-2019,-1049,-33730,-80
C00895=-2838,58294,-2009,-1048,-33734,-76
C00896=-2848,58304,-1994,-1046,-33740,-72
C00897=-2856,58318,-1974,-1045,-33748,-68
C00898=-2863,58333,-1950,-1044,-33757,-66
C00899=-2869,58350,-1925,-1043,-33767,-64
C00900=-2874,58367,-1900,-1042,-33778,-62
C00901=-2874,58387,-1869,-1042,-33790,-62
C00902=-2883,58398,-1854,-1040,-33796,-59
C00903=-2883,58398,-654,-1040,-33796,-59
C00904=-752,58146,-1001,-1326,-33648,-911
C00905=-752,58146,-2201,-1326,-33648,-911
C00906=-754,58143,-2205,-1325,-33646,-910
C00907=-756,58140,-2209,-1325,-33645,-909
C00908=-758,58138,-2213,-1325,-33643,-909
C00909=-759,58135,-2217,-1325,-33642,-908
C00910=-761,58133,-2221,-1325,-33640,-907
C00911=-762,58129,-2226,-1325,-33638,-907
C00912=-764,58127,-2230,-1324,-33636,-906
C00913=-765,58124,-2234,-1324,-33635,-905
C00914=-766,58121,-2239,-1324,-33633,-905
C00915=-766,58118,-2244,-1324,-33631,-905
C00916=-765,58114,-2250,-1324,-33628,-905
C00917=-765,58110,-2255,-1325,-33626,-905
C00918=-764,58107,-2260,-1325,-33624,-906
C00919=-762,58105,-2263,-1325,-33623,-906
C00920=-760,58103,-2266,-1325,-33622,-907
C00921=-758,58103,-2267,-1326,-33621,-908
C00922=-756,58101,-2269,-1326,-33621,-909
C00923=-754,58101,-2270,-1326,-33620,-910
C00924=-752,58102,-2267,-1326,-33621,-911
C00925=-750,58104,-2265,-1327,-33622,-911
C00926=-748,58106,-2261,-1327,-33624,-912
C00927=-746,58108,-2259,-1327,-33625,-913
C00928=-744,58110,-2255,-1327,-33626,-914
C00929=-742,58112,-2253,-1328,-33627,-915
C00930=-740,58114,-2249,-1328,-33628,-915
C00931=-739,58117,-2245,-1328,-33630,-916
C00932=-738,58120,-2240,-1328,-33632,-916
C00933=-736,58122,-2236,-1328,-33634,-917
C00934=-734,58125,-2232,-1328,-33635,-918
C00935=-734,58129,-2227,-1328,-33638,-918
C00936=-735,58132,-2222,-1328,-33640,-918
C00937=-737,58134,-2219,-1328,-33641,-917
C00938=-739,58135,-2217,-1328,-33641,-916
C00939=-741,58135,-2217,-1327,-33642,-915
C00940=-744,58135,-2217,-1327,-33642,-914
C00941=-746,58137,-2214,-1327,-33643,-913
C00942=-747,58139,-2211,-1326,-33644,-913
C00943=-748,58143,-2206,-1326,-33646,-912
C00944=-750,58145,-2201,-1326,-33648,-912
C00945=-752,58146,-2201,-1326,-33648,-911
C00946=-752,58146,-1001,-1326,-33648,-911
C00947=-2839,57899,-1405,-1054,-33494,-70
C00948=-2839,57899,-2605,-1054,-33494,-70
C00949=-2818,57878,-2637,-1057,-33481,-79
C00950=-2797,57849,-2680,-1060,-33464,-86
C00951=-2777,57821,-2723,-1063,-33446,-94
C00952=-2757,57792,-2767,-1066,-33429,-102
C00953=-2735,57767,-2804,-1069,-33413,-110
C00954=-2714,57741,-2843,-1073,-33398,-119
C00955=-2692,57717,-2879,-1076,-33383,-127
C00956=-2670,57693,-2915,-1079,-33369,-136
C00957=-2649,57667,-2954,-1082,-33353,-144
C00958=-2627,57641,-2993,-1086,-33337,-152
C00959=-2606,57615,-3032,-1089,-33321,-160
C00960=-2585,57587,-3074,-1092,-33304,-168
C00961=-2570,57557,-3120,-1095,-33285,-174
C00962=-2589,57527,-3166,-1093,-33267,-166
C00963=-2609,57498,-3209,-1090,-33250,-158
C00964=-2631,57471,-3250,-1088,-33233,-149
C00965=-2652,57447,-3287,-1085,-33219,-140
C00966=-2674,57422,-3325,-1083,-33203,-130
C00967=-2697,57400,-3358,-1080,-33190,-121
C00968=-2720,57378,-3392,-1077,-33177,-112
C00969=-2743,57356,-3425,-1075,-33164,-102
C00970=-2765,57331,-3464,-1072,-33148,-93
C00971=-2787,57304,-3504,-1070,-33132,-84
C00972=-2807,57275,-3548,-1067,-33115,-76
C00973=-2829,57248,-3588,-1065,-33099,-67
C00974=-2833,57289,-3526,-1064,-33124,-65
C00975=-2832,57334,-3459,-1063,-33151,-66
C00976=-2831,57378,-3393,-1063,-33177,-67
C00977=-2831,57422,-3326,-1062,-33204,-68
C00978=-2832,57467,-3258,-1061,-33231,-68
C00979=-2832,57511,-3191,-1060,-33258,-68
C00980=-2834,57555,-3126,-1060,-33285,-68
C00981=-2835,57597,-3062,-1059,-33310,-68
C00982=-2837,57639,-2998,-1058,-33336,-68
C00983=-2837,57683,-2931,-1057,-33363,-68
C00984=-2837,57728,-2864,-1056,-33390,-69
C00985=-2839,57772,-2798,-1056,-33416,-69
C00986=-2838,57814,-2735,-1055,-33442,-70
C00987=-2838,57855,-2673,-1054,-33467,-70
C00988=-2839,57899,-2605,-1054,-33494,-70
C00989=-2839,57899,-1405,-1054,-33494,-70
C00990=-2862,57865,-1458,-1051,-33473,-61
C00991=-2862,57865,-2658,-1051,-33473,-61
C00992=-2854,57831,-2709,-1053,-33452,-64
C00993=-2854,57785,-2778,-1053,-33425,-63
C00994=-2852,57740,-2846,-1054,-33397,-63
C00995=-2852,57694,-2915,-1055,-33369,-63
C00996=-2850,57649,-2983,-1056,-33342,-63
C00997=-2849,57604,-3051,-1057,-33315,-63
C00998=-2847,57559,-3120,-1058,-33287,-63
C00999=-2847,57513,-3189,-1058,-33259,-62
C01000=-2847,57467,-3258,-1059,-33232,-62
C01001=-2846,57421,-3327,-1060,-33204,-62
C01002=-2845,57376,-3395,-1061,-33176,-62
C01003=-2846,57330,-3466,-1061,-33148,-61
C01004=-2847,57285,-3533,-1062,-33121,-60
C01005=-2849,57243,-3596,-1062,-33096,-58
C01006=-2873,57264,-3565,-1059,-33108,-49
C01007=-2896,57287,-3530,-1055,-33123,-40
C01008=-2920,57306,-3501,-1052,-33134,-31
C01009=-2944,57324,-3475,-1048,-33145,-21
C01010=-2969,57341,-3449,-1045,-33156,-11
C01011=-2995,57356,-3427,-1041,-33165,-1
C01012=-3019,57375,-3399,-1038,-33176,8
C01013=-3043,57394,-3371,-1034,-33187,18
C01014=-3068,57411,-3345,-1031,-33198,27
C01015=-3092,57430,-3316,-1027,-33210,37
C01016=-3115,57453,-3282,-1024,-33224,46
C01017=-3138,57476,-3247,-1020,-33238,55
C01018=-3143,57503,-3206,-1019,-33254,56
C01019=-3121,57533,-3161,-1022,-33272,47
C01020=-3101,57563,-3116,-1024,-33290,39
C01021=-3079,57589,-3077,-1026,-33306,29
C01022=-3056,57615,-3037,-1029,-33322,20
C01023=-3033,57638,-3002,-1032,-33336,10
C01024=-3010,57663,-2964,-1035,-33351,1
C01025=-2987,57691,-2922,-1037,-33367,-8
C01026=-2965,57717,-2882,-1040,-33383,-18
C01027=-2942,57744,-2840,-1042,-33400,-27
C01028=-2921,57773,-2797,-1045,-33417,-36
C01029=-2901,57803,-2752,-1047,-33435,-44
C01030=-2881,57834,-2705,-1049,-33454,-53
C01031=-2862,57865,-2658,-1051,-33473,-61
C01032=-2862,57865,-1458,-1051,-33473,-61
C01033=-2751,59247,631,-1045,-34312,-122
C01034=-2751,59247,-569,-1045,-34312,-122
C01035=-2957,59244,-579,-1018,-34309,-39
C01036=-3131,59075,-836,-997,-34205,33
C01037=-3218,58778,-1285,-990,-34026,72
C01038=-3210,58445,-1787,-996,-33824,72
C01039=-3094,58170,-2200,-1016,-33658,29
C01040=-2904,58046,-2385,-1043,-33583,-46
C01041=-2923,57799,-2758,-1044,-33433,-36
C01042=-3093,57596,-3066,-1024,-33310,35
C01043=-3093,57405,-3354,-1027,-33195,37
C01044=-2907,57266,-3562,-1054,-33110,-35
C01045=-2993,57104,-3808,-1045,-33012,1
C01046=-3104,56999,-3966,-1032,-32949,46
C01047=-2917,57140,-3752,-1055,-33033,-30
C01048=-2845,56966,-4014,-1067,-32927,-57
C01049=-2899,56649,-4493,-1065,-32735,-31
C01050=-2976,56343,-4955,-1059,-32550,3
C01051=-3023,56066,-5373,-1057,-32383,25
C01052=-2955,56378,-4902,-1061,-32571,-6
C01053=-2876,56683,-4443,-1067,-32755,-41
C01054=-2788,56748,-4343,-1078,-32795,-77
C01055=-2707,56447,-4798,-1094,-32611,-105
C01056=-2609,56156,-5238,-1111,-32433,-141
C01057=-2564,56078,-5356,-1119,-32385,-158
C01058=-2663,56367,-4919,-1101,-32562,-122
C01059=-2749,56666,-4468,-1085,-32744,-91
C01060=-2829,56958,-4027,-1069,-32922,-63
C01061=-2765,57176,-3698,-1075,-33054,-91
C01062=-2560,57102,-3807,-1103,-33008,-172
C01063=-2548,57123,-3775,-1104,-33021,-177
C01064=-2753,57197,-3665,-1076,-33067,-96
C01065=-2701,57375,-3396,-1080,-33175,-119
C01066=-2548,57581,-3083,-1097,-33300,-183
C01067=-2718,57775,-2791,-1072,-33419,-117
C01068=-2834,58016,-2429,-1052,-33565,-74
C01069=-2624,58053,-2370,-1080,-33588,-159
C01070=-2462,58254,-2064,-1098,-33710,-226
C01071=-2385,58557,-1604,-1103,-33895,-261
C01072=-2426,58878,-1119,-1093,-34091,-248
C01073=-2557,59137,-730,-1072,-34247,-199
C01074=-2751,59247,-569,-1045,-34312,-122
C01075=-2751,59247,631,-1045,-34312,-122
//INST
///DATE 2026/04/22 17:00
///ATTR SC,RW
///GROUP1 RB1
NOP
MOVJ C00000 VJ=0.78
MOVJ C00001 VJ=0.78
MOVJ C00002 VJ=0.78
MOVL C00003 V=10.0
MOVL C00004 V=10.0
MOVL C00005 V=10.0
MOVL C00006 V=10.0
MOVL C00007 V=10.0
MOVL C00008 V=10.0
MOVL C00009 V=10.0
MOVL C00010 V=10.0
MOVL C00011 V=10.0
MOVL C00012 V=10.0
MOVL C00013 V=10.0
MOVL C00014 V=10.0
MOVL C00015 V=10.0
MOVL C00016 V=10.0
MOVL C00017 V=10.0
MOVL C00018 V=10.0
MOVL C00019 V=10.0
MOVL C00020 V=10.0
MOVL C00021 V=10.0
MOVL C00022 V=10.0
MOVL C00023 V=10.0
MOVL C00024 V=10.0
MOVL C00025 V=10.0
MOVL C00026 V=10.0
MOVL C00027 V=10.0
MOVL C00028 V=10.0
MOVL C00029 V=10.0
MOVL C00030 V=10.0
MOVL C00031 V=10.0
MOVL C00032 V=10.0
MOVL C00033 V=10.0
MOVL C00034 V=10.0
MOVL C00035 V=10.0
MOVL C00036 V=10.0
MOVL C00037 V=10.0
MOVL C00038 V=10.0
MOVL C00039 V=10.0
MOVL C00040 V=10.0
MOVL C00041 V=10.0
MOVL C00042 V=10.0
MOVJ C00043 VJ=0.78
MOVJ C00044 VJ=0.78
MOVJ C00045 VJ=0.78
MOVL C00046 V=10.0
MOVL C00047 V=10.0
MOVL C00048 V=10.0
MOVL C00049 V=10.0
MOVL C00050 V=10.0
MOVL C00051 V=10.0
MOVL C00052 V=10.0
MOVL C00053 V=10.0
MOVL C00054 V=10.0
MOVL C00055 V=10.0
MOVL C00056 V=10.0
MOVL C00057 V=10.0
MOVL C00058 V=10.0
MOVL C00059 V=10.0
MOVL C00060 V=10.0
MOVL C00061 V=10.0
MOVL C00062 V=10.0
MOVL C00063 V=10.0
MOVL C00064 V=10.0
MOVL C00065 V=10.0
MOVL C00066 V=10.0
MOVL C00067 V=10.0
MOVL C00068 V=10.0
MOVL C00069 V=10.0
MOVL C00070 V=10.0
MOVL C00071 V=10.0
MOVL C00072 V=10.0
MOVL C00073 V=10.0
MOVL C00074 V=10.0
MOVL C00075 V=10.0
MOVL C00076 V=10.0
MOVL C00077 V=10.0
MOVL C00078 V=10.0
MOVL C00079 V=10.0
MOVL C00080 V=10.0
MOVL C00081 V=10.0
MOVL C00082 V=10.0
MOVL C00083 V=10.0
MOVL C00084 V=10.0
MOVL C00085 V=10.0
MOVJ C00086 VJ=0.78
MOVJ C00087 VJ=0.78
MOVJ C00088 VJ=0.78
MOVL C00089 V=10.0
MOVL C00090 V=10.0
MOVL C00091 V=10.0
MOVL C00092 V=10.0
MOVL C00093 V=10.0
MOVL C00094 V=10.0
MOVL C00095 V=10.0
MOVL C00096 V=10.0
MOVL C00097 V=10.0
MOVL C00098 V=10.0
MOVL C00099 V=10.0
MOVL C00100 V=10.0
MOVL C00101 V=10.0
MOVL C00102 V=10.0
MOVL C00103 V=10.0
MOVL C00104 V=10.0
MOVL C00105 V=10.0
MOVL C00106 V=10.0
MOVL C00107 V=10.0
MOVL C00108 V=10.0
MOVL C00109 V=10.0
MOVL C00110 V=10.0
MOVL C00111 V=10.0
MOVL C00112 V=10.0
MOVL C00113 V=10.0
MOVL C00114 V=10.0
MOVL C00115 V=10.0
MOVL C00116 V=10.0
MOVL C00117 V=10.0
MOVL C00118 V=10.0
MOVL C00119 V=10.0
MOVL C00120 V=10.0
MOVL C00121 V=10.0
MOVL C00122 V=10.0
MOVL C00123 V=10.0
MOVL C00124 V=10.0
MOVL C00125 V=10.0
MOVL C00126 V=10.0
MOVL C00127 V=10.0
MOVL C00128 V=10.0
MOVJ C00129 VJ=0.78
MOVJ C00130 VJ=0.78
MOVJ C00131 VJ=0.78
MOVL C00132 V=10.0
MOVL C00133 V=10.0
MOVL C00134 V=10.0
MOVL C00135 V=10.0
MOVL C00136 V=10.0
MOVL C00137 V=10.0
MOVL C00138 V=10.0
MOVL C00139 V=10.0
MOVL C00140 V=10.0
MOVL C00141 V=10.0
MOVL C00142 V=10.0
MOVL C00143 V=10.0
MOVL C00144 V=10.0
MOVL C00145 V=10.0
MOVL C00146 V=10.0
MOVL C00147 V=10.0
MOVL C00148 V=10.0
MOVL C00149 V=10.0
MOVL C00150 V=10.0
MOVL C00151 V=10.0
MOVL C00152 V=10.0
MOVL C00153 V=10.0
MOVL C00154 V=10.0
MOVL C00155 V=10.0
MOVL C00156 V=10.0
MOVL C00157 V=10.0
MOVL C00158 V=10.0
MOVL C00159 V=10.0
MOVL C00160 V=10.0
MOVL C00161 V=10.0
MOVL C00162 V=10.0
MOVL C00163 V=10.0
MOVL C00164 V=10.0
MOVL C00165 V=10.0
MOVL C00166 V=10.0
MOVL C00167 V=10.0
MOVL C00168 V=10.0
MOVL C00169 V=10.0
MOVL C00170 V=10.0
MOVL C00171 V=10.0
MOVJ C00172 VJ=0.78
MOVJ C00173 VJ=0.78
MOVJ C00174 VJ=0.78
MOVL C00175 V=10.0
MOVL C00176 V=10.0
MOVL C00177 V=10.0
MOVL C00178 V=10.0
MOVL C00179 V=10.0
MOVL C00180 V=10.0
MOVL C00181 V=10.0
MOVL C00182 V=10.0
MOVL C00183 V=10.0
MOVL C00184 V=10.0
MOVL C00185 V=10.0
MOVL C00186 V=10.0
MOVL C00187 V=10.0
MOVL C00188 V=10.0
MOVL C00189 V=10.0
MOVL C00190 V=10.0
MOVL C00191 V=10.0
MOVL C00192 V=10.0
MOVL C00193 V=10.0
MOVL C00194 V=10.0
MOVL C00195 V=10.0
MOVL C00196 V=10.0
MOVL C00197 V=10.0
MOVL C00198 V=10.0
MOVL C00199 V=10.0
MOVL C00200 V=10.0
MOVL C00201 V=10.0
MOVL C00202 V=10.0
MOVL C00203 V=10.0
MOVL C00204 V=10.0
MOVL C00205 V=10.0
MOVL C00206 V=10.0
MOVL C00207 V=10.0
MOVL C00208 V=10.0
MOVL C00209 V=10.0
MOVL C00210 V=10.0
MOVL C00211 V=10.0
MOVL C00212 V=10.0
MOVL C00213 V=10.0
MOVL C00214 V=10.0
MOVJ C00215 VJ=0.78
MOVJ C00216 VJ=0.78
MOVJ C00217 VJ=0.78
MOVL C00218 V=10.0
MOVL C00219 V=10.0
MOVL C00220 V=10.0
MOVL C00221 V=10.0
MOVL C00222 V=10.0
MOVL C00223 V=10.0
MOVL C00224 V=10.0
MOVL C00225 V=10.0
MOVL C00226 V=10.0
MOVL C00227 V=10.0
MOVL C00228 V=10.0
MOVL C00229 V=10.0
MOVL C00230 V=10.0
MOVL C00231 V=10.0
MOVL C00232 V=10.0
MOVL C00233 V=10.0
MOVL C00234 V=10.0
MOVL C00235 V=10.0
MOVL C00236 V=10.0
MOVL C00237 V=10.0
MOVL C00238 V=10.0
MOVL C00239 V=10.0
MOVL C00240 V=10.0
MOVL C00241 V=10.0
MOVL C00242 V=10.0
MOVL C00243 V=10.0
MOVL C00244 V=10.0
MOVL C00245 V=10.0
MOVL C00246 V=10.0
MOVL C00247 V=10.0
MOVL C00248 V=10.0
MOVL C00249 V=10.0
MOVL C00250 V=10.0
MOVL C00251 V=10.0
MOVL C00252 V=10.0
MOVL C00253 V=10.0
MOVL C00254 V=10.0
MOVL C00255 V=10.0
MOVL C00256 V=10.0
MOVL C00257 V=10.0
MOVJ C00258 VJ=0.78
MOVJ C00259 VJ=0.78
MOVJ C00260 VJ=0.78
MOVL C00261 V=10.0
MOVL C00262 V=10.0
MOVL C00263 V=10.0
MOVL C00264 V=10.0
MOVL C00265 V=10.0
MOVL C00266 V=10.0
MOVL C00267 V=10.0
MOVL C00268 V=10.0
MOVL C00269 V=10.0
MOVL C00270 V=10.0
MOVL C00271 V=10.0
MOVL C00272 V=10.0
MOVL C00273 V=10.0
MOVL C00274 V=10.0
MOVL C00275 V=10.0
MOVL C00276 V=10.0
MOVL C00277 V=10.0
MOVL C00278 V=10.0
MOVL C00279 V=10.0
MOVL C00280 V=10.0
MOVL C00281 V=10.0
MOVL C00282 V=10.0
MOVL C00283 V=10.0
MOVL C00284 V=10.0
MOVL C00285 V=10.0
MOVL C00286 V=10.0
MOVL C00287 V=10.0
MOVL C00288 V=10.0
MOVL C00289 V=10.0
MOVL C00290 V=10.0
MOVL C00291 V=10.0
MOVL C00292 V=10.0
MOVL C00293 V=10.0
MOVL C00294 V=10.0
MOVL C00295 V=10.0
MOVL C00296 V=10.0
MOVL C00297 V=10.0
MOVL C00298 V=10.0
MOVL C00299 V=10.0
MOVL C00300 V=10.0
MOVJ C00301 VJ=0.78
MOVJ C00302 VJ=0.78
MOVJ C00303 VJ=0.78
MOVL C00304 V=10.0
MOVL C00305 V=10.0
MOVL C00306 V=10.0
MOVL C00307 V=10.0
MOVL C00308 V=10.0
MOVL C00309 V=10.0
MOVL C00310 V=10.0
MOVL C00311 V=10.0
MOVL C00312 V=10.0
MOVL C00313 V=10.0
MOVL C00314 V=10.0
MOVL C00315 V=10.0
MOVL C00316 V=10.0
MOVL C00317 V=10.0
MOVL C00318 V=10.0
MOVL C00319 V=10.0
MOVL C00320 V=10.0
MOVL C00321 V=10.0
MOVL C00322 V=10.0
MOVL C00323 V=10.0
MOVL C00324 V=10.0
MOVL C00325 V=10.0
MOVL C00326 V=10.0
MOVL C00327 V=10.0
MOVL C00328 V=10.0
MOVL C00329 V=10.0
MOVL C00330 V=10.0
MOVL C00331 V=10.0
MOVL C00332 V=10.0
MOVL C00333 V=10.0
MOVL C00334 V=10.0
MOVL C00335 V=10.0
MOVL C00336 V=10.0
MOVL C00337 V=10.0
MOVL C00338 V=10.0
MOVL C00339 V=10.0
MOVL C00340 V=10.0
MOVL C00341 V=10.0
MOVL C00342 V=10.0
MOVL C00343 V=10.0
MOVJ C00344 VJ=0.78
MOVJ C00345 VJ=0.78
MOVJ C00346 VJ=0.78
MOVL C00347 V=10.0
MOVL C00348 V=10.0
MOVL C00349 V=10.0
MOVL C00350 V=10.0
MOVL C00351 V=10.0
MOVL C00352 V=10.0
MOVL C00353 V=10.0
MOVL C00354 V=10.0
MOVL C00355 V=10.0
MOVL C00356 V=10.0
MOVL C00357 V=10.0
MOVL C00358 V=10.0
MOVL C00359 V=10.0
MOVL C00360 V=10.0
MOVL C00361 V=10.0
MOVL C00362 V=10.0
MOVL C00363 V=10.0
MOVL C00364 V=10.0
MOVL C00365 V=10.0
MOVL C00366 V=10.0
MOVL C00367 V=10.0
MOVL C00368 V=10.0
MOVL C00369 V=10.0
MOVL C00370 V=10.0
MOVL C00371 V=10.0
MOVL C00372 V=10.0
MOVL C00373 V=10.0
MOVL C00374 V=10.0
MOVL C00375 V=10.0
MOVL C00376 V=10.0
MOVL C00377 V=10.0
MOVL C00378 V=10.0
MOVL C00379 V=10.0
MOVL C00380 V=10.0
MOVL C00381 V=10.0
MOVL C00382 V=10.0
MOVL C00383 V=10.0
MOVL C00384 V=10.0
MOVL C00385 V=10.0
MOVL C00386 V=10.0
MOVJ C00387 VJ=0.78
MOVJ C00388 VJ=0.78
MOVJ C00389 VJ=0.78
MOVL C00390 V=10.0
MOVL C00391 V=10.0
MOVL C00392 V=10.0
MOVL C00393 V=10.0
MOVL C00394 V=10.0
MOVL C00395 V=10.0
MOVL C00396 V=10.0
MOVL C00397 V=10.0
MOVL C00398 V=10.0
MOVL C00399 V=10.0
MOVL C00400 V=10.0
MOVL C00401 V=10.0
MOVL C00402 V=10.0
MOVL C00403 V=10.0
MOVL C00404 V=10.0
MOVL C00405 V=10.0
MOVL C00406 V=10.0
MOVL C00407 V=10.0
MOVL C00408 V=10.0
MOVL C00409 V=10.0
MOVL C00410 V=10.0
MOVL C00411 V=10.0
MOVL C00412 V=10.0
MOVL C00413 V=10.0
MOVL C00414 V=10.0
MOVL C00415 V=10.0
MOVL C00416 V=10.0
MOVL C00417 V=10.0
MOVL C00418 V=10.0
MOVL C00419 V=10.0
MOVL C00420 V=10.0
MOVL C00421 V=10.0
MOVL C00422 V=10.0
MOVL C00423 V=10.0
MOVL C00424 V=10.0
MOVL C00425 V=10.0
MOVL C00426 V=10.0
MOVL C00427 V=10.0
MOVL C00428 V=10.0
MOVL C00429 V=10.0
MOVJ C00430 VJ=0.78
MOVJ C00431 VJ=0.78
MOVJ C00432 VJ=0.78
MOVL C00433 V=10.0
MOVL C00434 V=10.0
MOVL C00435 V=10.0
MOVL C00436 V=10.0
MOVL C00437 V=10.0
MOVL C00438 V=10.0
MOVL C00439 V=10.0
MOVL C00440 V=10.0
MOVL C00441 V=10.0
MOVL C00442 V=10.0
MOVL C00443 V=10.0
MOVL C00444 V=10.0
MOVL C00445 V=10.0
MOVL C00446 V=10.0
MOVL C00447 V=10.0
MOVL C00448 V=10.0
MOVL C00449 V=10.0
MOVL C00450 V=10.0
MOVL C00451 V=10.0
MOVL C00452 V=10.0
MOVL C00453 V=10.0
MOVL C00454 V=10.0
MOVL C00455 V=10.0
MOVL C00456 V=10.0
MOVL C00457 V=10.0
MOVL C00458 V=10.0
MOVL C00459 V=10.0
MOVL C00460 V=10.0
MOVL C00461 V=10.0
MOVL C00462 V=10.0
MOVL C00463 V=10.0
MOVL C00464 V=10.0
MOVL C00465 V=10.0
MOVL C00466 V=10.0
MOVL C00467 V=10.0
MOVL C00468 V=10.0
MOVL C00469 V=10.0
MOVL C00470 V=10.0
MOVL C00471 V=10.0
MOVL C00472 V=10.0
MOVJ C00473 VJ=0.78
MOVJ C00474 VJ=0.78
MOVJ C00475 VJ=0.78
MOVL C00476 V=10.0
MOVL C00477 V=10.0
MOVL C00478 V=10.0
MOVL C00479 V=10.0
MOVL C00480 V=10.0
MOVL C00481 V=10.0
MOVL C00482 V=10.0
MOVL C00483 V=10.0
MOVL C00484 V=10.0
MOVL C00485 V=10.0
MOVL C00486 V=10.0
MOVL C00487 V=10.0
MOVL C00488 V=10.0
MOVL C00489 V=10.0
MOVL C00490 V=10.0
MOVL C00491 V=10.0
MOVL C00492 V=10.0
MOVL C00493 V=10.0
MOVL C00494 V=10.0
MOVL C00495 V=10.0
MOVL C00496 V=10.0
MOVL C00497 V=10.0
MOVL C00498 V=10.0
MOVL C00499 V=10.0
MOVL C00500 V=10.0
MOVL C00501 V=10.0
MOVL C00502 V=10.0
MOVL C00503 V=10.0
MOVL C00504 V=10.0
MOVL C00505 V=10.0
MOVL C00506 V=10.0
MOVL C00507 V=10.0
MOVL C00508 V=10.0
MOVL C00509 V=10.0
MOVL C00510 V=10.0
MOVL C00511 V=10.0
MOVL C00512 V=10.0
MOVL C00513 V=10.0
MOVL C00514 V=10.0
MOVL C00515 V=10.0
MOVJ C00516 VJ=0.78
MOVJ C00517 VJ=0.78
MOVJ C00518 VJ=0.78
MOVL C00519 V=10.0
MOVL C00520 V=10.0
MOVL C00521 V=10.0
MOVL C00522 V=10.0
MOVL C00523 V=10.0
MOVL C00524 V=10.0
MOVL C00525 V=10.0
MOVL C00526 V=10.0
MOVL C00527 V=10.0
MOVL C00528 V=10.0
MOVL C00529 V=10.0
MOVL C00530 V=10.0
MOVL C00531 V=10.0
MOVL C00532 V=10.0
MOVL C00533 V=10.0
MOVL C00534 V=10.0
MOVL C00535 V=10.0
MOVL C00536 V=10.0
MOVL C00537 V=10.0
MOVL C00538 V=10.0
MOVL C00539 V=10.0
MOVL C00540 V=10.0
MOVL C00541 V=10.0
MOVL C00542 V=10.0
MOVL C00543 V=10.0
MOVL C00544 V=10.0
MOVL C00545 V=10.0
MOVL C00546 V=10.0
MOVL C00547 V=10.0
MOVL C00548 V=10.0
MOVL C00549 V=10.0
MOVL C00550 V=10.0
MOVL C00551 V=10.0
MOVL C00552 V=10.0
MOVL C00553 V=10.0
MOVL C00554 V=10.0
MOVL C00555 V=10.0
MOVL C00556 V=10.0
MOVL C00557 V=10.0
MOVL C00558 V=10.0
MOVJ C00559 VJ=0.78
MOVJ C00560 VJ=0.78
MOVJ C00561 VJ=0.78
MOVL C00562 V=10.0
MOVL C00563 V=10.0
MOVL C00564 V=10.0
MOVL C00565 V=10.0
MOVL C00566 V=10.0
MOVL C00567 V=10.0
MOVL C00568 V=10.0
MOVL C00569 V=10.0
MOVL C00570 V=10.0
MOVL C00571 V=10.0
MOVL C00572 V=10.0
MOVL C00573 V=10.0
MOVL C00574 V=10.0
MOVL C00575 V=10.0
MOVL C00576 V=10.0
MOVL C00577 V=10.0
MOVL C00578 V=10.0
MOVL C00579 V=10.0
MOVL C00580 V=10.0
MOVL C00581 V=10.0
MOVL C00582 V=10.0
MOVL C00583 V=10.0
MOVL C00584 V=10.0
MOVL C00585 V=10.0
MOVL C00586 V=10.0
MOVL C00587 V=10.0
MOVL C00588 V=10.0
MOVL C00589 V=10.0
MOVL C00590 V=10.0
MOVL C00591 V=10.0
MOVL C00592 V=10.0
MOVL C00593 V=10.0
MOVL C00594 V=10.0
MOVL C00595 V=10.0
MOVL C00596 V=10.0
MOVL C00597 V=10.0
MOVL C00598 V=10.0
MOVL C00599 V=10.0
MOVL C00600 V=10.0
MOVL C00601 V=10.0
MOVJ C00602 VJ=0.78
MOVJ C00603 VJ=0.78
MOVJ C00604 VJ=0.78
MOVL C00605 V=10.0
MOVL C00606 V=10.0
MOVL C00607 V=10.0
MOVL C00608 V=10.0
MOVL C00609 V=10.0
MOVL C00610 V=10.0
MOVL C00611 V=10.0
MOVL C00612 V=10.0
MOVL C00613 V=10.0
MOVL C00614 V=10.0
MOVL C00615 V=10.0
MOVL C00616 V=10.0
MOVL C00617 V=10.0
MOVL C00618 V=10.0
MOVL C00619 V=10.0
MOVL C00620 V=10.0
MOVL C00621 V=10.0
MOVL C00622 V=10.0
MOVL C00623 V=10.0
MOVL C00624 V=10.0
MOVL C00625 V=10.0
MOVL C00626 V=10.0
MOVL C00627 V=10.0
MOVL C00628 V=10.0
MOVL C00629 V=10.0
MOVL C00630 V=10.0
MOVL C00631 V=10.0
MOVL C00632 V=10.0
MOVL C00633 V=10.0
MOVL C00634 V=10.0
MOVL C00635 V=10.0
MOVL C00636 V=10.0
MOVL C00637 V=10.0
MOVL C00638 V=10.0
MOVL C00639 V=10.0
MOVL C00640 V=10.0
MOVL C00641 V=10.0
MOVL C00642 V=10.0
MOVL C00643 V=10.0
MOVL C00644 V=10.0
MOVJ C00645 VJ=0.78
MOVJ C00646 VJ=0.78
MOVJ C00647 VJ=0.78
MOVL C00648 V=10.0
MOVL C00649 V=10.0
MOVL C00650 V=10.0
MOVL C00651 V=10.0
MOVL C00652 V=10.0
MOVL C00653 V=10.0
MOVL C00654 V=10.0
MOVL C00655 V=10.0
MOVL C00656 V=10.0
MOVL C00657 V=10.0
MOVL C00658 V=10.0
MOVL C00659 V=10.0
MOVL C00660 V=10.0
MOVL C00661 V=10.0
MOVL C00662 V=10.0
MOVL C00663 V=10.0
MOVL C00664 V=10.0
MOVL C00665 V=10.0
MOVL C00666 V=10.0
MOVL C00667 V=10.0
MOVL C00668 V=10.0
MOVL C00669 V=10.0
MOVL C00670 V=10.0
MOVL C00671 V=10.0
MOVL C00672 V=10.0
MOVL C00673 V=10.0
MOVL C00674 V=10.0
MOVL C00675 V=10.0
MOVL C00676 V=10.0
MOVL C00677 V=10.0
MOVL C00678 V=10.0
MOVL C00679 V=10.0
MOVL C00680 V=10.0
MOVL C00681 V=10.0
MOVL C00682 V=10.0
MOVL C00683 V=10.0
MOVL C00684 V=10.0
MOVL C00685 V=10.0
MOVL C00686 V=10.0
MOVL C00687 V=10.0
MOVJ C00688 VJ=0.78
MOVJ C00689 VJ=0.78
MOVJ C00690 VJ=0.78
MOVL C00691 V=10.0
MOVL C00692 V=10.0
MOVL C00693 V=10.0
MOVL C00694 V=10.0
MOVL C00695 V=10.0
MOVL C00696 V=10.0
MOVL C00697 V=10.0
MOVL C00698 V=10.0
MOVL C00699 V=10.0
MOVL C00700 V=10.0
MOVL C00701 V=10.0
MOVL C00702 V=10.0
MOVL C00703 V=10.0
MOVL C00704 V=10.0
MOVL C00705 V=10.0
MOVL C00706 V=10.0
MOVL C00707 V=10.0
MOVL C00708 V=10.0
MOVL C00709 V=10.0
MOVL C00710 V=10.0
MOVL C00711 V=10.0
MOVL C00712 V=10.0
MOVL C00713 V=10.0
MOVL C00714 V=10.0
MOVL C00715 V=10.0
MOVL C00716 V=10.0
MOVL C00717 V=10.0
MOVL C00718 V=10.0
MOVL C00719 V=10.0
MOVL C00720 V=10.0
MOVL C00721 V=10.0
MOVL C00722 V=10.0
MOVL C00723 V=10.0
MOVL C00724 V=10.0
MOVL C00725 V=10.0
MOVL C00726 V=10.0
MOVL C00727 V=10.0
MOVL C00728 V=10.0
MOVL C00729 V=10.0
MOVL C00730 V=10.0
MOVJ C00731 VJ=0.78
MOVJ C00732 VJ=0.78
MOVJ C00733 VJ=0.78
MOVL C00734 V=10.0
MOVL C00735 V=10.0
MOVL C00736 V=10.0
MOVL C00737 V=10.0
MOVL C00738 V=10.0
MOVL C00739 V=10.0
MOVL C00740 V=10.0
MOVL C00741 V=10.0
MOVL C00742 V=10.0
MOVL C00743 V=10.0
MOVL C00744 V=10.0
MOVL C00745 V=10.0
MOVL C00746 V=10.0
MOVL C00747 V=10.0
MOVL C00748 V=10.0
MOVL C00749 V=10.0
MOVL C00750 V=10.0
MOVL C00751 V=10.0
MOVL C00752 V=10.0
MOVL C00753 V=10.0
MOVL C00754 V=10.0
MOVL C00755 V=10.0
MOVL C00756 V=10.0
MOVL C00757 V=10.0
MOVL C00758 V=10.0
MOVL C00759 V=10.0
MOVL C00760 V=10.0
MOVL C00761 V=10.0
MOVL C00762 V=10.0
MOVL C00763 V=10.0
MOVL C00764 V=10.0
MOVL C00765 V=10.0
MOVL C00766 V=10.0
MOVL C00767 V=10.0
MOVL C00768 V=10.0
MOVL C00769 V=10.0
MOVL C00770 V=10.0
MOVL C00771 V=10.0
MOVL C00772 V=10.0
MOVL C00773 V=10.0
MOVJ C00774 VJ=0.78
MOVJ C00775 VJ=0.78
MOVJ C00776 VJ=0.78
MOVL C00777 V=10.0
MOVL C00778 V=10.0
MOVL C00779 V=10.0
MOVL C00780 V=10.0
MOVL C00781 V=10.0
MOVL C00782 V=10.0
MOVL C00783 V=10.0
MOVL C00784 V=10.0
MOVL C00785 V=10.0
MOVL C00786 V=10.0
MOVL C00787 V=10.0
MOVL C00788 V=10.0
MOVL C00789 V=10.0
MOVL C00790 V=10.0
MOVL C00791 V=10.0
MOVL C00792 V=10.0
MOVL C00793 V=10.0
MOVL C00794 V=10.0
MOVL C00795 V=10.0
MOVL C00796 V=10.0
MOVL C00797 V=10.0
MOVL C00798 V=10.0
MOVL C00799 V=10.0
MOVL C00800 V=10.0
MOVL C00801 V=10.0
MOVL C00802 V=10.0
MOVL C00803 V=10.0
MOVL C00804 V=10.0
MOVL C00805 V=10.0
MOVL C00806 V=10.0
MOVL C00807 V=10.0
MOVL C00808 V=10.0
MOVL C00809 V=10.0
MOVL C00810 V=10.0
MOVL C00811 V=10.0
MOVL C00812 V=10.0
MOVL C00813 V=10.0
MOVL C00814 V=10.0
MOVL C00815 V=10.0
MOVL C00816 V=10.0
MOVJ C00817 VJ=0.78
MOVJ C00818 VJ=0.78
MOVJ C00819 VJ=0.78
MOVL C00820 V=10.0
MOVL C00821 V=10.0
MOVL C00822 V=10.0
MOVL C00823 V=10.0
MOVL C00824 V=10.0
MOVL C00825 V=10.0
MOVL C00826 V=10.0
MOVL C00827 V=10.0
MOVL C00828 V=10.0
MOVL C00829 V=10.0
MOVL C00830 V=10.0
MOVL C00831 V=10.0
MOVL C00832 V=10.0
MOVL C00833 V=10.0
MOVL C00834 V=10.0
MOVL C00835 V=10.0
MOVL C00836 V=10.0
MOVL C00837 V=10.0
MOVL C00838 V=10.0
MOVL C00839 V=10.0
MOVL C00840 V=10.0
MOVL C00841 V=10.0
MOVL C00842 V=10.0
MOVL C00843 V=10.0
MOVL C00844 V=10.0
MOVL C00845 V=10.0
MOVL C00846 V=10.0
MOVL C00847 V=10.0
MOVL C00848 V=10.0
MOVL C00849 V=10.0
MOVL C00850 V=10.0
MOVL C00851 V=10.0
MOVL C00852 V=10.0
MOVL C00853 V=10.0
MOVL C00854 V=10.0
MOVL C00855 V=10.0
MOVL C00856 V=10.0
MOVL C00857 V=10.0
MOVL C00858 V=10.0
MOVL C00859 V=10.0
MOVJ C00860 VJ=0.78
MOVJ C00861 VJ=0.78
MOVJ C00862 VJ=0.78
MOVL C00863 V=10.0
MOVL C00864 V=10.0
MOVL C00865 V=10.0
MOVL C00866 V=10.0
MOVL C00867 V=10.0
MOVL C00868 V=10.0
MOVL C00869 V=10.0
MOVL C00870 V=10.0
MOVL C00871 V=10.0
MOVL C00872 V=10.0
MOVL C00873 V=10.0
MOVL C00874 V=10.0
MOVL C00875 V=10.0
MOVL C00876 V=10.0
MOVL C00877 V=10.0
MOVL C00878 V=10.0
MOVL C00879 V=10.0
MOVL C00880 V=10.0
MOVL C00881 V=10.0
MOVL C00882 V=10.0
MOVL C00883 V=10.0
MOVL C00884 V=10.0
MOVL C00885 V=10.0
MOVL C00886 V=10.0
MOVL C00887 V=10.0
MOVL C00888 V=10.0
MOVL C00889 V=10.0
MOVL C00890 V=10.0
MOVL C00891 V=10.0
MOVL C00892 V=10.0
MOVL C00893 V=10.0
MOVL C00894 V=10.0
MOVL C00895 V=10.0
MOVL C00896 V=10.0
MOVL C00897 V=10.0
MOVL C00898 V=10.0
MOVL C00899 V=10.0
MOVL C00900 V=10.0
MOVL C00901 V=10.0
MOVL C00902 V=10.0
MOVJ C00903 VJ=0.78
MOVJ C00904 VJ=0.78
MOVJ C00905 VJ=0.78
MOVL C00906 V=10.0
MOVL C00907 V=10.0
MOVL C00908 V=10.0
MOVL C00909 V=10.0
MOVL C00910 V=10.0
MOVL C00911 V=10.0
MOVL C00912 V=10.0
MOVL C00913 V=10.0
MOVL C00914 V=10.0
MOVL C00915 V=10.0
MOVL C00916 V=10.0
MOVL C00917 V=10.0
MOVL C00918 V=10.0
MOVL C00919 V=10.0
MOVL C00920 V=10.0
MOVL C00921 V=10.0
MOVL C00922 V=10.0
MOVL C00923 V=10.0
MOVL C00924 V=10.0
MOVL C00925 V=10.0
MOVL C00926 V=10.0
MOVL C00927 V=10.0
MOVL C00928 V=10.0
MOVL C00929 V=10.0
MOVL C00930 V=10.0
MOVL C00931 V=10.0
MOVL C00932 V=10.0
MOVL C00933 V=10.0
MOVL C00934 V=10.0
MOVL C00935 V=10.0
MOVL C00936 V=10.0
MOVL C00937 V=10.0
MOVL C00938 V=10.0
MOVL C00939 V=10.0
MOVL C00940 V=10.0
MOVL C00941 V=10.0
MOVL C00942 V=10.0
MOVL C00943 V=10.0
MOVL C00944 V=10.0
MOVL C00945 V=10.0
MOVJ C00946 VJ=0.78
MOVJ C00947 VJ=0.78
MOVJ C00948 VJ=0.78
MOVL C00949 V=10.0
MOVL C00950 V=10.0
MOVL C00951 V=10.0
MOVL C00952 V=10.0
MOVL C00953 V=10.0
MOVL C00954 V=10.0
MOVL C00955 V=10.0
MOVL C00956 V=10.0
MOVL C00957 V=10.0
MOVL C00958 V=10.0
MOVL C00959 V=10.0
MOVL C00960 V=10.0
MOVL C00961 V=10.0
MOVL C00962 V=10.0
MOVL C00963 V=10.0
MOVL C00964 V=10.0
MOVL C00965 V=10.0
MOVL C00966 V=10.0
MOVL C00967 V=10.0
MOVL C00968 V=10.0
MOVL C00969 V=10.0
MOVL C00970 V=10.0
MOVL C00971 V=10.0
MOVL C00972 V=10.0
MOVL C00973 V=10.0
MOVL C00974 V=10.0
MOVL C00975 V=10.0
MOVL C00976 V=10.0
MOVL C00977 V=10.0
MOVL C00978 V=10.0
MOVL C00979 V=10.0
MOVL C00980 V=10.0
MOVL C00981 V=10.0
MOVL C00982 V=10.0
MOVL C00983 V=10.0
MOVL C00984 V=10.0
MOVL C00985 V=10.0
MOVL C00986 V=10.0
MOVL C00987 V=10.0
MOVL C00988 V=10.0
MOVJ C00989 VJ=0.78
MOVJ C00990 VJ=0.78
MOVJ C00991 VJ=0.78
MOVL C00992 V=10.0
MOVL C00993 V=10.0
MOVL C00994 V=10.0
MOVL C00995 V=10.0
MOVL C00996 V=10.0
MOVL C00997 V=10.0
MOVL C00998 V=10.0
MOVL C00999 V=10.0
MOVL C01000 V=10.0
MOVL C01001 V=10.0
MOVL C01002 V=10.0
MOVL C01003 V=10.0
MOVL C01004 V=10.0
MOVL C01005 V=10.0
MOVL C01006 V=10.0
MOVL C01007 V=10.0
MOVL C01008 V=10.0
MOVL C01009 V=10.0
MOVL C01010 V=10.0
MOVL C01011 V=10.0
MOVL C01012 V=10.0
MOVL C01013 V=10.0
MOVL C01014 V=10.0
MOVL C01015 V=10.0
MOVL C01016 V=10.0
MOVL C01017 V=10.0
MOVL C01018 V=10.0
MOVL C01019 V=10.0
MOVL C01020 V=10.0
MOVL C01021 V=10.0
MOVL C01022 V=10.0
MOVL C01023 V=10.0
MOVL C01024 V=10.0
MOVL C01025 V=10.0
MOVL C01026 V=10.0
MOVL C01027 V=10.0
MOVL C01028 V=10.0
MOVL C01029 V=10.0
MOVL C01030 V=10.0
MOVL C01031 V=10.0
MOVJ C01032 VJ=0.78
MOVJ C01033 VJ=0.78
MOVJ C01034 VJ=0.78
MOVL C01035 V=10.0
MOVL C01036 V=10.0
MOVL C01037 V=10.0
MOVL C01038 V=10.0
MOVL C01039 V=10.0
MOVL C01040 V=10.0
MOVL C01041 V=10.0
MOVL C01042 V=10.0
MOVL C01043 V=10.0
MOVL C01044 V=10.0
MOVL C01045 V=10.0
MOVL C01046 V=10.0
MOVL C01047 V=10.0
MOVL C01048 V=10.0
MOVL C01049 V=10.0
MOVL C01050 V=10.0
MOVL C01051 V=10.0
MOVL C01052 V=10.0
MOVL C01053 V=10.0
MOVL C01054 V=10.0
MOVL C01055 V=10.0
MOVL C01056 V=10.0
MOVL C01057 V=10.0
MOVL C01058 V=10.0
MOVL C01059 V=10.0
MOVL C01060 V=10.0
MOVL C01061 V=10.0
MOVL C01062 V=10.0
MOVL C01063 V=10.0
MOVL C01064 V=10.0
MOVL C01065 V=10.0
MOVL C01066 V=10.0
MOVL C01067 V=10.0
MOVL C01068 V=10.0
MOVL C01069 V=10.0
MOVL C01070 V=10.0
MOVL C01071 V=10.0
MOVL C01072 V=10.0
MOVL C01073 V=10.0
MOVL C01074 V=10.0
MOVJ C01075 VJ=0.78
END
